LIN {X 0,Y 424.985,Z 1036.91,A -85,B 0,C 180,E1 -9892.159,E2 -9892.159} C_VEL
LIN {X 0,Y 424.826,Z 1042.69,A -85,B 0,C 180,E1 -9893.35,E2 -9893.35} C_VEL
LIN {X 0,Y 424.561,Z 1046.489,A -85,B 0,C 180,E1 -9894.3,E2 -9894.3} C_VEL
LIN {X 0,Y 424.338,Z 1049.56,A -85,B 0,C 180,E1 -9895.25,E2 -9895.25} C_VEL
LIN {X 0,Y 424.395,Z 1051.936,A -85,B 0,C 180,E1 -9896.202,E2 -9896.202} C_VEL
LIN {X 0,Y 424.27,Z 1053.752,A -85,B 0,C 180,E1 -9897.152,E2 -9897.152} C_VEL
LIN {X 0,Y 424.174,Z 1055.045,A -85,B 0,C 180,E1 -9898.101,E2 -9898.101} C_VEL
LIN {X 0,Y 424.113,Z 1055.839,A -85,B 0,C 180,E1 -9899.051,E2 -9899.051} C_VEL
LIN {X 0,Y 424.106,Z 1056.112,A -85,B 0,C 180,E1 -9900,E2 -9900} C_VEL
LIN {X 0,Y 424.112,Z 1055.78,A -85,B 0,C 180,E1 -9900.95,E2 -9900.95} C_VEL
LIN {X 0,Y 424.165,Z 1054.937,A -85,B 0,C 180,E1 -9901.899,E2 -9901.899} C_VEL
LIN {X 0,Y 424.262,Z 1053.59,A -85,B 0,C 180,E1 -9902.849,E2 -9902.849} C_VEL
LIN {X 0,Y 424.316,Z 1050.534,A -85,B 0,C 180,E1 -9904.275,E2 -9904.275} C_VEL
LIN {X 0,Y 424.525,Z 1046.159,A -85,B 0,C 180,E1 -9905.701,E2 -9905.701} C_VEL
LIN {X 0,Y 424.759,Z 1040.098,A -85,B 0,C 180,E1 -9907.128,E2 -9907.128} C_VEL
LIN {X 0,Y 424.953,Z 1035.048,A -85,B 0,C 180,E1 -9908.082,E2 -9908.082} C_VEL
LIN {X 0,Y 425.243,Z 1028.948,A -85,B 0,C 180,E1 -9909.034,E2 -9909.034} C_VEL
LIN {X 0,Y 425.687,Z 1020.492,A -85,B 0,C 180,E1 -9910.103,E2 -9910.103} C_VEL
LIN {X 0,Y 426.165,Z 1011.11,A -85,B 0,C 180,E1 -9911.053,E2 -9911.053} C_VEL
LIN {X 0,Y 426.592,Z 1000.255,A -85,B 0,C 180,E1 -9911.885,E2 -9911.885} C_VEL
LIN {X 0,Y 426.862,Z 991.105,A -85,B 0,C 180,E1 -9912.42,E2 -9912.42} C_VEL
LIN {X 0,Y 427.087,Z 981.57,A -85,B 0,C 180,E1 -9912.836,E2 -9912.836} C_VEL
LIN {X 0,Y 427.334,Z 971.535,A -85,B 0,C 180,E1 -9913.131,E2 -9913.131} C_VEL
LIN {X 0,Y 427.866,Z 911.953,A -85,B 0,C 180,E1 -9914.276,E2 -9914.276} C_VEL
LIN {X 0,Y 425.344,Z 897.558,A -85,B 0,C 180,E1 -9914.656,E2 -9914.656} C_VEL
LIN {X 0,Y 425.733,Z 888.265,A -85,B 0,C 180,E1 -9917.287,E2 -9917.287} C_VEL
LIN {X 0,Y 425.456,Z 882.672,A -85,B 0,C 180,E1 -9918.916,E2 -9918.916} C_VEL
LIN {X 0,Y 425.385,Z 882.313,A -85,B 0,C 180,E1 -9919.045,E2 -9919.045} C_VEL
LIN {X 0,Y 425.286,Z 882.318,A -85,B 0,C 180,E1 -9922.339,E2 -9922.339} C_VEL
LIN {X 0,Y 425.25,Z 882.327,A -85,B 0,C 180,E1 -9925.449,E2 -9925.449} C_VEL
LIN {X 0,Y 425.297,Z 882.318,A -85,B 0,C 180,E1 -9928.858,E2 -9928.858} C_VEL
LIN {X 0,Y 425.254,Z 882.324,A -85,B 0,C 180,E1 -9931.929,E2 -9931.929} C_VEL
LIN {X 0,Y 425.294,Z 882.32,A -85,B 0,C 180,E1 -9935.337,E2 -9935.337} C_VEL
LIN {X 0,Y 425.275,Z 882.319,A -85,B 0,C 180,E1 -9938.902,E2 -9938.902} C_VEL
LIN {X 0,Y 425.256,Z 882.322,A -85,B 0,C 180,E1 -9942.656,E2 -9942.656} C_VEL
LIN {X 0,Y 425.285,Z 882.318,A -85,B 0,C 180,E1 -9945.284,E2 -9945.284} C_VEL
LIN {X 0,Y 425.247,Z 882.326,A -85,B 0,C 180,E1 -9948.618,E2 -9948.618} C_VEL
LIN {X 0,Y 425.27,Z 882.326,A -85,B 0,C 180,E1 -9952.305,E2 -9952.305} C_VEL
LIN {X 0,Y 425.288,Z 882.318,A -85,B 0,C 180,E1 -9955.816,E2 -9955.816} C_VEL
LIN {X 0,Y 425.288,Z 882.319,A -85,B 0,C 180,E1 -9959.241,E2 -9959.241} C_VEL
LIN {X 0,Y 425.24,Z 882.326,A -85,B 0,C 180,E1 -9962.435,E2 -9962.435} C_VEL
LIN {X 0,Y 425.319,Z 882.315,A -85,B 0,C 180,E1 -9965.6,E2 -9965.6} C_VEL
LIN {X 0,Y 425.286,Z 882.32,A -85,B 0,C 180,E1 -9968.681,E2 -9968.681} C_VEL
LIN {X 0,Y 425.3,Z 882.318,A -85,B 0,C 180,E1 -9971.701,E2 -9971.701} C_VEL
LIN {X 0,Y 425.324,Z 882.314,A -85,B 0,C 180,E1 -9974.67,E2 -9974.67} C_VEL
LIN {X 0,Y 425.411,Z 882.309,A -85,B 0,C 180,E1 -9977.598,E2 -9977.598} C_VEL
LIN {X 0,Y 425.398,Z 882.308,A -85,B 0,C 180,E1 -9981.449,E2 -9981.449} C_VEL
LIN {X 0,Y 425.497,Z 882.293,A -85,B 0,C 180,E1 -9984.377,E2 -9984.377} C_VEL
LIN {X 0,Y 425.564,Z 882.289,A -85,B 0,C 180,E1 -9988.107,E2 -9988.107} C_VEL
LIN {X 0,Y 425.495,Z 882.293,A -85,B 0,C 180,E1 -9988.519,E2 -9988.519} C_VEL
LIN {X 0,Y 424.768,Z 882.383,A -85,B 0,C 180,E1 -9989.308,E2 -9989.308} C_VEL
LIN {X 0,Y 421.933,Z 882.737,A -85,B 0,C 180,E1 -9990.592,E2 -9990.592} C_VEL
LIN {X 0,Y 419.57,Z 883.031,A -85,B 0,C 180,E1 -9991.629,E2 -9991.629} C_VEL
LIN {X 0,Y 418.55,Z 883.161,A -85,B 0,C 180,E1 -9992.429,E2 -9992.429} C_VEL
LIN {X 0,Y 418.461,Z 883.168,A -85,B 0,C 180,E1 -9992.7,E2 -9992.7} C_VEL
LIN {X 0,Y 418.473,Z 883.168,A -85,B 0,C 180,E1 -9995.784,E2 -9995.784} C_VEL
LIN {X 0,Y 418.37,Z 883.184,A -85,B 0,C 180,E1 -9998.696,E2 -9998.696} C_VEL
LIN {X 0,Y 418.357,Z 883.188,A -85,B 0,C 180,E1 -10002.615,E2 -10002.615} C_VEL
LIN {X 0,Y 418.284,Z 883.195,A -85,B 0,C 180,E1 -10006.597,E2 -10006.597} C_VEL
LIN {X 0,Y 418.247,Z 883.195,A -85,B 0,C 180,E1 -10009.779,E2 -10009.779} C_VEL
LIN {X 0,Y 418.228,Z 883.2,A -85,B 0,C 180,E1 -10012.737,E2 -10012.737} C_VEL
LIN {X 0,Y 418.213,Z 883.199,A -85,B 0,C 180,E1 -10015.908,E2 -10015.908} C_VEL
LIN {X 0,Y 418.259,Z 883.198,A -85,B 0,C 180,E1 -10019.163,E2 -10019.163} C_VEL
LIN {X 0,Y 418.235,Z 883.196,A -85,B 0,C 180,E1 -10022.529,E2 -10022.529} C_VEL
LIN {X 0,Y 418.251,Z 883.195,A -85,B 0,C 180,E1 -10024.842,E2 -10024.842} C_VEL
LIN {X 0,Y 418.235,Z 883.197,A -85,B 0,C 180,E1 -10028.444,E2 -10028.444} C_VEL
LIN {X 0,Y 418.221,Z 883.202,A -85,B 0,C 180,E1 -10032.236,E2 -10032.236} C_VEL
LIN {X 0,Y 418.238,Z 883.196,A -85,B 0,C 180,E1 -10035.108,E2 -10035.108} C_VEL
LIN {X 0,Y 418.221,Z 883.2,A -85,B 0,C 180,E1 -10037.764,E2 -10037.764} C_VEL
LIN {X 0,Y 418.23,Z 883.197,A -85,B 0,C 180,E1 -10041.555,E2 -10041.555} C_VEL
LIN {X 0,Y 418.253,Z 883.195,A -85,B 0,C 180,E1 -10045.158,E2 -10045.158} C_VEL
LIN {X 0,Y 418.242,Z 883.195,A -85,B 0,C 180,E1 -10047.471,E2 -10047.471} C_VEL
LIN {X 0,Y 418.261,Z 883.199,A -85,B 0,C 180,E1 -10050.898,E2 -10050.898} C_VEL
LIN {X 0,Y 418.213,Z 883.199,A -85,B 0,C 180,E1 -10054.092,E2 -10054.092} C_VEL
LIN {X 0,Y 418.235,Z 883.198,A -85,B 0,C 180,E1 -10057.552,E2 -10057.552} C_VEL
LIN {X 0,Y 418.255,Z 883.194,A -85,B 0,C 180,E1 -10060.362,E2 -10060.362} C_VEL
LIN {X 0,Y 418.283,Z 883.197,A -85,B 0,C 180,E1 -10063.403,E2 -10063.403} C_VEL
LIN {X 0,Y 418.355,Z 883.187,A -85,B 0,C 180,E1 -10067.385,E2 -10067.385} C_VEL
LIN {X 0,Y 418.369,Z 883.182,A -85,B 0,C 180,E1 -10071.304,E2 -10071.304} C_VEL
LIN {X 0,Y 418.471,Z 883.169,A -85,B 0,C 180,E1 -10074.216,E2 -10074.216} C_VEL
LIN {X 0,Y 418.53,Z 883.165,A -85,B 0,C 180,E1 -10078.075,E2 -10078.075} C_VEL
LIN {X 0,Y 418.408,Z 883.175,A -85,B 0,C 180,E1 -10080.962,E2 -10080.962} C_VEL
LIN {X 0,Y 418.454,Z 883.169,A -85,B 0,C 180,E1 -10082.888,E2 -10082.888} C_VEL
LIN {X 0,Y 418.47,Z 883.168,A -85,B 0,C 180,E1 -10085.783,E2 -10085.783} C_VEL
LIN {X 0,Y 418.368,Z 883.184,A -85,B 0,C 180,E1 -10088.695,E2 -10088.695} C_VEL
LIN {X 0,Y 418.354,Z 883.189,A -85,B 0,C 180,E1 -10092.614,E2 -10092.614} C_VEL
LIN {X 0,Y 418.281,Z 883.195,A -85,B 0,C 180,E1 -10096.596,E2 -10096.596} C_VEL
LIN {X 0,Y 418.244,Z 883.195,A -85,B 0,C 180,E1 -10099.779,E2 -10099.779} C_VEL
LIN {X 0,Y 418.224,Z 883.201,A -85,B 0,C 180,E1 -10102.737,E2 -10102.737} C_VEL
LIN {X 0,Y 418.209,Z 883.2,A -85,B 0,C 180,E1 -10105.908,E2 -10105.908} C_VEL
LIN {X 0,Y 418.255,Z 883.199,A -85,B 0,C 180,E1 -10109.162,E2 -10109.162} C_VEL
LIN {X 0,Y 418.23,Z 883.197,A -85,B 0,C 180,E1 -10112.529,E2 -10112.529} C_VEL
LIN {X 0,Y 418.247,Z 883.195,A -85,B 0,C 180,E1 -10114.842,E2 -10114.842} C_VEL
LIN {X 0,Y 418.23,Z 883.197,A -85,B 0,C 180,E1 -10118.444,E2 -10118.444} C_VEL
LIN {X 0,Y 418.216,Z 883.202,A -85,B 0,C 180,E1 -10122.236,E2 -10122.236} C_VEL
LIN {X 0,Y 418.233,Z 883.196,A -85,B 0,C 180,E1 -10125.108,E2 -10125.108} C_VEL
LIN {X 0,Y 418.216,Z 883.201,A -85,B 0,C 180,E1 -10127.763,E2 -10127.763} C_VEL
LIN {X 0,Y 418.225,Z 883.198,A -85,B 0,C 180,E1 -10131.555,E2 -10131.555} C_VEL
LIN {X 0,Y 418.248,Z 883.195,A -85,B 0,C 180,E1 -10135.158,E2 -10135.158} C_VEL
LIN {X 0,Y 418.238,Z 883.196,A -85,B 0,C 180,E1 -10137.471,E2 -10137.471} C_VEL
LIN {X 0,Y 418.256,Z 883.199,A -85,B 0,C 180,E1 -10140.898,E2 -10140.898} C_VEL
LIN {X 0,Y 418.258,Z 883.255,A -85,B 0,C 180,E1 -10144.411,E2 -10144.411} C_VEL
LIN {X 0,Y 420.166,Z 893.538,A -85,B 0,C 180,E1 -10146.921,E2 -10146.921} C_VEL
LIN {X 0,Y 419.942,Z 901.074,A -85,B 0,C 180,E1 -10148.654,E2 -10148.654} C_VEL
LIN {X 0,Y 419.121,Z 915.553,A -85,B 0,C 180,E1 -10151.928,E2 -10151.928} C_VEL
LIN {X 0,Y 418.376,Z 930.113,A -85,B 0,C 180,E1 -10155.141,E2 -10155.141} C_VEL
LIN {X 0,Y 420.95,Z 951.978,A -85,B 0,C 180,E1 -10155.663,E2 -10155.663} C_VEL
LIN {X 0,Y 420.299,Z 1007.525,A -85,B 0,C 180,E1 -10156.769,E2 -10156.769} C_VEL
LIN {X 0,Y 419.904,Z 1018.346,A -85,B 0,C 180,E1 -10157.125,E2 -10157.125} C_VEL
LIN {X 0,Y 419.54,Z 1029.214,A -85,B 0,C 180,E1 -10157.667,E2 -10157.667} C_VEL
LIN {X 0,Y 419.115,Z 1039.643,A -85,B 0,C 180,E1 -10158.391,E2 -10158.391} C_VEL
LIN {X 0,Y 418.722,Z 1047.891,A -85,B 0,C 180,E1 -10159.116,E2 -10159.116} C_VEL
LIN {X 0,Y 418.32,Z 1055.741,A -85,B 0,C 180,E1 -10159.962,E2 -10159.962} C_VEL
LIN {X 0,Y 417.897,Z 1063.972,A -85,B 0,C 180,E1 -10161.05,E2 -10161.05} C_VEL
LIN {X 0,Y 417.593,Z 1071.163,A -85,B 0,C 180,E1 -10162.262,E2 -10162.262} C_VEL
LIN {X 0,Y 417.341,Z 1076.904,A -85,B 0,C 180,E1 -10163.49,E2 -10163.49} C_VEL
LIN {X 0,Y 417.213,Z 1081.322,A -85,B 0,C 180,E1 -10164.684,E2 -10164.684} C_VEL
LIN {X 0,Y 417.114,Z 1084.17,A -85,B 0,C 180,E1 -10165.651,E2 -10165.651} C_VEL
LIN {X 0,Y 417.086,Z 1087.252,A -85,B 0,C 180,E1 -10167.102,E2 -10167.102} C_VEL
LIN {X 0,Y 417.073,Z 1088.619,A -85,B 0,C 180,E1 -10168.068,E2 -10168.068} C_VEL
LIN {X 0,Y 417.029,Z 1089.473,A -85,B 0,C 180,E1 -10169.034,E2 -10169.034} C_VEL
LIN {X 0,Y 417.023,Z 1089.769,A -85,B 0,C 180,E1 -10170,E2 -10170} C_VEL
LIN {X 0,Y 417.029,Z 1089.463,A -85,B 0,C 180,E1 -10170.965,E2 -10170.965} C_VEL
LIN {X 0,Y 417.073,Z 1088.655,A -85,B 0,C 180,E1 -10171.931,E2 -10171.931} C_VEL
LIN {X 0,Y 417.082,Z 1087.336,A -85,B 0,C 180,E1 -10172.897,E2 -10172.897} C_VEL
LIN {X 0,Y 417.114,Z 1084.266,A -85,B 0,C 180,E1 -10174.348,E2 -10174.348} C_VEL
LIN {X 0,Y 417.214,Z 1081.472,A -85,B 0,C 180,E1 -10175.316,E2 -10175.316} C_VEL
LIN {X 0,Y 417.342,Z 1077.084,A -85,B 0,C 180,E1 -10176.511,E2 -10176.511} C_VEL
LIN {X 0,Y 417.524,Z 1072.603,A -85,B 0,C 180,E1 -10177.496,E2 -10177.496} C_VEL
LIN {X 0,Y 417.725,Z 1067.312,A -85,B 0,C 180,E1 -10178.465,E2 -10178.465} C_VEL
LIN {X 0,Y 418.117,Z 1060.957,A -85,B 0,C 180,E1 -10179.432,E2 -10179.432} C_VEL
LIN {X 0,Y 418.516,Z 1053.237,A -85,B 0,C 180,E1 -10180.4,E2 -10180.4} C_VEL
LIN {X 0,Y 419.023,Z 1043.686,A -85,B 0,C 180,E1 -10181.366,E2 -10181.366} C_VEL
LIN {X 0,Y 419.428,Z 1034.458,A -85,B 0,C 180,E1 -10182.09,E2 -10182.09} C_VEL
LIN {X 0,Y 419.811,Z 1024.464,A -85,B 0,C 180,E1 -10182.693,E2 -10182.693} C_VEL
LIN {X 0,Y 420.227,Z 1015.136,A -85,B 0,C 180,E1 -10183.11,E2 -10183.11} C_VEL
LIN {X 0,Y 420.542,Z 1005.59,A -85,B 0,C 180,E1 -10183.407,E2 -10183.407} C_VEL
LIN {X 0,Y 421.166,Z 949.616,A -85,B 0,C 180,E1 -10184.57,E2 -10184.57} C_VEL
LIN {X 0,Y 418.931,Z 931.747,A -85,B 0,C 180,E1 -10185.066,E2 -10185.066} C_VEL
LIN {X 0,Y 418.429,Z 928.431,A -85,B 0,C 180,E1 -10185.177,E2 -10185.177} C_VEL
LIN {X 0,Y 419.239,Z 913.478,A -85,B 0,C 180,E1 -10188.573,E2 -10188.573} C_VEL
LIN {X 0,Y 420.175,Z 899.489,A -85,B 0,C 180,E1 -10191.849,E2 -10191.849} C_VEL
LIN {X 0,Y 420.291,Z 894.287,A -85,B 0,C 180,E1 -10193.119,E2 -10193.119} C_VEL
LIN {X 0,Y 418.805,Z 885.701,A -85,B 0,C 180,E1 -10195.403,E2 -10195.403} C_VEL
LIN {X 0,Y 418.244,Z 883.203,A -85,B 0,C 180,E1 -10196.174,E2 -10196.174} C_VEL
LIN {X 0,Y 418.252,Z 883.202,A -85,B 0,C 180,E1 -10199.163,E2 -10199.163} C_VEL
LIN {X 0,Y 418.246,Z 883.202,A -85,B 0,C 180,E1 -10202.842,E2 -10202.842} C_VEL
LIN {X 0,Y 418.235,Z 883.199,A -85,B 0,C 180,E1 -10206.236,E2 -10206.236} C_VEL
LIN {X 0,Y 418.19,Z 883.208,A -85,B 0,C 180,E1 -10209.689,E2 -10209.689} C_VEL
LIN {X 0,Y 418.203,Z 883.204,A -85,B 0,C 180,E1 -10212.318,E2 -10212.318} C_VEL
LIN {X 0,Y 418.232,Z 883.199,A -85,B 0,C 180,E1 -10215.108,E2 -10215.108} C_VEL
LIN {X 0,Y 418.214,Z 883.203,A -85,B 0,C 180,E1 -10217.764,E2 -10217.764} C_VEL
LIN {X 0,Y 418.224,Z 883.201,A -85,B 0,C 180,E1 -10221.555,E2 -10221.555} C_VEL
LIN {X 0,Y 418.247,Z 883.197,A -85,B 0,C 180,E1 -10225.158,E2 -10225.158} C_VEL
LIN {X 0,Y 418.237,Z 883.199,A -85,B 0,C 180,E1 -10227.472,E2 -10227.472} C_VEL
LIN {X 0,Y 418.255,Z 883.2,A -85,B 0,C 180,E1 -10230.899,E2 -10230.899} C_VEL
LIN {X 0,Y 418.207,Z 883.204,A -85,B 0,C 180,E1 -10234.092,E2 -10234.092} C_VEL
LIN {X 0,Y 418.229,Z 883.206,A -85,B 0,C 180,E1 -10237.553,E2 -10237.553} C_VEL
LIN {X 0,Y 418.265,Z 883.342,A -85,B 0,C 180,E1 -10239.689,E2 -10239.689} C_VEL
LIN {X 0,Y 419.149,Z 888.393,A -85,B 0,C 180,E1 -10241.423,E2 -10241.423} C_VEL
LIN {X 0,Y 419.053,Z 894.734,A -85,B 0,C 180,E1 -10243.435,E2 -10243.435} C_VEL
LIN {X 0,Y 418.734,Z 899.597,A -85,B 0,C 180,E1 -10244.928,E2 -10244.928} C_VEL
LIN {X 0,Y 421.443,Z 912.992,A -85,B 0,C 180,E1 -10245.358,E2 -10245.358} C_VEL
LIN {X 0,Y 420.863,Z 963.311,A -85,B 0,C 180,E1 -10246.415,E2 -10246.415} C_VEL
LIN {X 0,Y 420.498,Z 978.918,A -85,B 0,C 180,E1 -10246.776,E2 -10246.776} C_VEL
LIN {X 0,Y 420.228,Z 990.494,A -85,B 0,C 180,E1 -10247.259,E2 -10247.259} C_VEL
LIN {X 0,Y 419.889,Z 998.061,A -85,B 0,C 180,E1 -10247.678,E2 -10247.678} C_VEL
LIN {X 0,Y 419.592,Z 1006.59,A -85,B 0,C 180,E1 -10248.283,E2 -10248.283} C_VEL
LIN {X 0,Y 419.251,Z 1014.804,A -85,B 0,C 180,E1 -10249.008,E2 -10249.008} C_VEL
LIN {X 0,Y 418.832,Z 1022.619,A -85,B 0,C 180,E1 -10249.852,E2 -10249.852} C_VEL
LIN {X 0,Y 418.373,Z 1029.936,A -85,B 0,C 180,E1 -10250.818,E2 -10250.818} C_VEL
LIN {X 0,Y 417.969,Z 1037.324,A -85,B 0,C 180,E1 -10252.027,E2 -10252.027} C_VEL
LIN {X 0,Y 417.763,Z 1043.07,A -85,B 0,C 180,E1 -10253.238,E2 -10253.238} C_VEL
LIN {X 0,Y 417.527,Z 1046.849,A -85,B 0,C 180,E1 -10254.204,E2 -10254.204} C_VEL
LIN {X 0,Y 417.272,Z 1049.911,A -85,B 0,C 180,E1 -10255.17,E2 -10255.17} C_VEL
LIN {X 0,Y 417.314,Z 1052.278,A -85,B 0,C 180,E1 -10256.138,E2 -10256.138} C_VEL
LIN {X 0,Y 417.21,Z 1054.083,A -85,B 0,C 180,E1 -10257.104,E2 -10257.104} C_VEL
LIN {X 0,Y 417.102,Z 1055.363,A -85,B 0,C 180,E1 -10258.069,E2 -10258.069} C_VEL
LIN {X 0,Y 417.034,Z 1056.141,A -85,B 0,C 180,E1 -10259.035,E2 -10259.035} C_VEL
LIN {X 0,Y 417.025,Z 1056.403,A -85,B 0,C 180,E1 -10260,E2 -10260} C_VEL
LIN {X 0,Y 417.033,Z 1056.058,A -85,B 0,C 180,E1 -10260.966,E2 -10260.966} C_VEL
LIN {X 0,Y 417.093,Z 1055.187,A -85,B 0,C 180,E1 -10261.932,E2 -10261.932} C_VEL
LIN {X 0,Y 417.181,Z 1053.815,A -85,B 0,C 180,E1 -10262.897,E2 -10262.897} C_VEL
LIN {X 0,Y 417.226,Z 1050.717,A -85,B 0,C 180,E1 -10264.348,E2 -10264.348} C_VEL
LIN {X 0,Y 417.464,Z 1046.294,A -85,B 0,C 180,E1 -10265.798,E2 -10265.798} C_VEL
LIN {X 0,Y 417.697,Z 1040.156,A -85,B 0,C 180,E1 -10267.25,E2 -10267.25} C_VEL
LIN {X 0,Y 417.906,Z 1035.047,A -85,B 0,C 180,E1 -10268.219,E2 -10268.219} C_VEL
LIN {X 0,Y 418.233,Z 1028.882,A -85,B 0,C 180,E1 -10269.186,E2 -10269.186} C_VEL
LIN {X 0,Y 418.626,Z 1021.379,A -85,B 0,C 180,E1 -10270.153,E2 -10270.153} C_VEL
LIN {X 0,Y 419.071,Z 1013.359,A -85,B 0,C 180,E1 -10270.998,E2 -10270.998} C_VEL
LIN {X 0,Y 419.502,Z 1003.366,A -85,B 0,C 180,E1 -10271.843,E2 -10271.843} C_VEL
LIN {X 0,Y 419.796,Z 992.781,A -85,B 0,C 180,E1 -10272.509,E2 -10272.509} C_VEL
LIN {X 0,Y 420.046,Z 982.95,A -85,B 0,C 180,E1 -10272.963,E2 -10272.963} C_VEL
LIN {X 0,Y 420.314,Z 973.531,A -85,B 0,C 180,E1 -10273.262,E2 -10273.262} C_VEL
LIN {X 0,Y 420.965,Z 912.92,A -85,B 0,C 180,E1 -10274.463,E2 -10274.463} C_VEL
LIN {X 0,Y 418.335,Z 897.792,A -85,B 0,C 180,E1 -10274.876,E2 -10274.876} C_VEL
LIN {X 0,Y 418.721,Z 888.371,A -85,B 0,C 180,E1 -10277.586,E2 -10277.586} C_VEL
LIN {X 0,Y 418.349,Z 883.188,A -85,B 0,C 180,E1 -10279.187,E2 -10279.187} C_VEL
LIN {X 0,Y 418.225,Z 883.201,A -85,B 0,C 180,E1 -10282.738,E2 -10282.738} C_VEL
LIN {X 0,Y 418.21,Z 883.2,A -85,B 0,C 180,E1 -10285.909,E2 -10285.909} C_VEL
LIN {X 0,Y 418.256,Z 883.198,A -85,B 0,C 180,E1 -10289.163,E2 -10289.163} C_VEL
LIN {X 0,Y 418.25,Z 883.195,A -85,B 0,C 180,E1 -10292.842,E2 -10292.842} C_VEL
LIN {X 0,Y 418.24,Z 883.197,A -85,B 0,C 180,E1 -10296.237,E2 -10296.237} C_VEL
LIN {X 0,Y 418.199,Z 883.206,A -85,B 0,C 180,E1 -10299.689,E2 -10299.689} C_VEL
LIN {X 0,Y 418.207,Z 883.203,A -85,B 0,C 180,E1 -10302.318,E2 -10302.318} C_VEL
LIN {X 0,Y 418.236,Z 883.196,A -85,B 0,C 180,E1 -10305.109,E2 -10305.109} C_VEL
LIN {X 0,Y 418.219,Z 883.2,A -85,B 0,C 180,E1 -10307.764,E2 -10307.764} C_VEL
LIN {X 0,Y 418.229,Z 883.197,A -85,B 0,C 180,E1 -10311.556,E2 -10311.556} C_VEL
LIN {X 0,Y 418.252,Z 883.195,A -85,B 0,C 180,E1 -10315.158,E2 -10315.158} C_VEL
LIN {X 0,Y 418.242,Z 883.196,A -85,B 0,C 180,E1 -10317.472,E2 -10317.472} C_VEL
LIN {X 0,Y 418.26,Z 883.199,A -85,B 0,C 180,E1 -10320.899,E2 -10320.899} C_VEL
LIN {X 0,Y 418.213,Z 883.199,A -85,B 0,C 180,E1 -10324.092,E2 -10324.092} C_VEL
LIN {X 0,Y 418.228,Z 883.202,A -85,B 0,C 180,E1 -10327.263,E2 -10327.263} C_VEL
LIN {X 0,Y 418.255,Z 883.194,A -85,B 0,C 180,E1 -10330.363,E2 -10330.363} C_VEL
LIN {X 0,Y 418.33,Z 883.191,A -85,B 0,C 180,E1 -10333.405,E2 -10333.405} C_VEL
LIN {X 0,Y 418.357,Z 883.187,A -85,B 0,C 180,E1 -10337.386,E2 -10337.386} C_VEL
LIN {X 0,Y 418.37,Z 883.182,A -85,B 0,C 180,E1 -10341.304,E2 -10341.304} C_VEL
LIN {X 0,Y 418.473,Z 883.169,A -85,B 0,C 180,E1 -10344.217,E2 -10344.217} C_VEL
LIN {X 0,Y 418.532,Z 883.165,A -85,B 0,C 180,E1 -10348.076,E2 -10348.076} C_VEL
LIN {X 0,Y 418.41,Z 883.174,A -85,B 0,C 180,E1 -10350.963,E2 -10350.963} C_VEL
LIN {X 0,Y 418.461,Z 883.168,A -85,B 0,C 180,E1 -10352.7,E2 -10352.7} C_VEL
LIN {X 0,Y 417.781,Z 883.254,A -85,B 0,C 180,E1 -10353.502,E2 -10353.502} C_VEL
LIN {X 0,Y 414.933,Z 883.613,A -85,B 0,C 180,E1 -10354.806,E2 -10354.806} C_VEL
LIN {X 0,Y 412.524,Z 883.913,A -85,B 0,C 180,E1 -10355.859,E2 -10355.859} C_VEL
LIN {X 0,Y 411.482,Z 884.042,A -85,B 0,C 180,E1 -10356.672,E2 -10356.672} C_VEL
LIN {X 0,Y 411.391,Z 884.05,A -85,B 0,C 180,E1 -10356.948,E2 -10356.948} C_VEL
LIN {X 0,Y 411.276,Z 884.064,A -85,B 0,C 180,E1 -10359.839,E2 -10359.839} C_VEL
LIN {X 0,Y 411.31,Z 884.061,A -85,B 0,C 180,E1 -10363.103,E2 -10363.103} C_VEL
LIN {X 0,Y 411.214,Z 884.077,A -85,B 0,C 180,E1 -10366.891,E2 -10366.891} C_VEL
LIN {X 0,Y 411.209,Z 884.072,A -85,B 0,C 180,E1 -10369.988,E2 -10369.988} C_VEL
LIN {X 0,Y 411.179,Z 884.082,A -85,B 0,C 180,E1 -10373.149,E2 -10373.149} C_VEL
LIN {X 0,Y 411.167,Z 884.077,A -85,B 0,C 180,E1 -10376.386,E2 -10376.386} C_VEL
LIN {X 0,Y 411.196,Z 884.076,A -85,B 0,C 180,E1 -10379.713,E2 -10379.713} C_VEL
LIN {X 0,Y 411.207,Z 884.074,A -85,B 0,C 180,E1 -10383.156,E2 -10383.156} C_VEL
LIN {X 0,Y 411.191,Z 884.074,A -85,B 0,C 180,E1 -10386.551,E2 -10386.551} C_VEL
LIN {X 0,Y 411.17,Z 884.082,A -85,B 0,C 180,E1 -10389.72,E2 -10389.72} C_VEL
LIN {X 0,Y 411.164,Z 884.077,A -85,B 0,C 180,E1 -10393.135,E2 -10393.135} C_VEL
LIN {X 0,Y 411.167,Z 884.081,A -85,B 0,C 180,E1 -10395.882,E2 -10395.882} C_VEL
LIN {X 0,Y 411.159,Z 884.078,A -85,B 0,C 180,E1 -10399.492,E2 -10399.492} C_VEL
LIN {X 0,Y 411.18,Z 884.078,A -85,B 0,C 180,E1 -10402.024,E2 -10402.024} C_VEL
LIN {X 0,Y 411.205,Z 884.073,A -85,B 0,C 180,E1 -10405.123,E2 -10405.123} C_VEL
LIN {X 0,Y 411.163,Z 884.078,A -85,B 0,C 180,E1 -10408.002,E2 -10408.002} C_VEL
LIN {X 0,Y 411.171,Z 884.077,A -85,B 0,C 180,E1 -10411.406,E2 -10411.406} C_VEL
LIN {X 0,Y 411.191,Z 884.081,A -85,B 0,C 180,E1 -10414.941,E2 -10414.941} C_VEL
LIN {X 0,Y 411.203,Z 884.072,A -85,B 0,C 180,E1 -10417.913,E2 -10417.913} C_VEL
LIN {X 0,Y 411.193,Z 884.079,A -85,B 0,C 180,E1 -10421.049,E2 -10421.049} C_VEL
LIN {X 0,Y 411.202,Z 884.072,A -85,B 0,C 180,E1 -10424.129,E2 -10424.129} C_VEL
LIN {X 0,Y 411.305,Z 884.063,A -85,B 0,C 180,E1 -10427.165,E2 -10427.165} C_VEL
LIN {X 0,Y 411.274,Z 884.065,A -85,B 0,C 180,E1 -10430.16,E2 -10430.16} C_VEL
LIN {X 0,Y 411.393,Z 884.049,A -85,B 0,C 180,E1 -10433.131,E2 -10433.131} C_VEL
LIN {X 0,Y 411.283,Z 884.063,A -85,B 0,C 180,E1 -10435.098,E2 -10435.098} C_VEL
LIN {X 0,Y 411.499,Z 884.042,A -85,B 0,C 180,E1 -10438.042,E2 -10438.042} C_VEL
LIN {X 0,Y 411.378,Z 884.05,A -85,B 0,C 180,E1 -10440.978,E2 -10440.978} C_VEL
LIN {X 0,Y 411.413,Z 884.046,A -85,B 0,C 180,E1 -10442.937,E2 -10442.937} C_VEL
LIN {X 0,Y 411.418,Z 884.048,A -85,B 0,C 180,E1 -10445.882,E2 -10445.882} C_VEL
LIN {X 0,Y 411.307,Z 884.062,A -85,B 0,C 180,E1 -10448.846,E2 -10448.846} C_VEL
LIN {X 0,Y 411.271,Z 884.064,A -85,B 0,C 180,E1 -10451.833,E2 -10451.833} C_VEL
LIN {X 0,Y 411.212,Z 884.076,A -85,B 0,C 180,E1 -10454.854,E2 -10454.854} C_VEL
LIN {X 0,Y 411.204,Z 884.072,A -85,B 0,C 180,E1 -10457.917,E2 -10457.917} C_VEL
LIN {X 0,Y 411.188,Z 884.081,A -85,B 0,C 180,E1 -10461.034,E2 -10461.034} C_VEL
LIN {X 0,Y 411.172,Z 884.076,A -85,B 0,C 180,E1 -10464.218,E2 -10464.218} C_VEL
LIN {X 0,Y 411.141,Z 884.084,A -85,B 0,C 180,E1 -10467.486,E2 -10467.486} C_VEL
LIN {X 0,Y 411.192,Z 884.076,A -85,B 0,C 180,E1 -10469.713,E2 -10469.713} C_VEL
LIN {X 0,Y 411.203,Z 884.075,A -85,B 0,C 180,E1 -10473.156,E2 -10473.156} C_VEL
LIN {X 0,Y 411.187,Z 884.074,A -85,B 0,C 180,E1 -10476.551,E2 -10476.551} C_VEL
LIN {X 0,Y 411.166,Z 884.083,A -85,B 0,C 180,E1 -10479.719,E2 -10479.719} C_VEL
LIN {X 0,Y 411.16,Z 884.078,A -85,B 0,C 180,E1 -10483.135,E2 -10483.135} C_VEL
LIN {X 0,Y 411.163,Z 884.082,A -85,B 0,C 180,E1 -10485.881,E2 -10485.881} C_VEL
LIN {X 0,Y 411.155,Z 884.078,A -85,B 0,C 180,E1 -10489.492,E2 -10489.492} C_VEL
LIN {X 0,Y 411.176,Z 884.079,A -85,B 0,C 180,E1 -10492.024,E2 -10492.024} C_VEL
LIN {X 0,Y 411.2,Z 884.073,A -85,B 0,C 180,E1 -10495.123,E2 -10495.123} C_VEL
LIN {X 0,Y 411.158,Z 884.079,A -85,B 0,C 180,E1 -10498.002,E2 -10498.002} C_VEL
LIN {X 0,Y 411.166,Z 884.078,A -85,B 0,C 180,E1 -10501.406,E2 -10501.406} C_VEL
LIN {X 0,Y 411.25,Z 884.212,A -85,B 0,C 180,E1 -10504.267,E2 -10504.267} C_VEL
LIN {X 0,Y 413.189,Z 895.116,A -85,B 0,C 180,E1 -10506.97,E2 -10506.97} C_VEL
LIN {X 0,Y 412.837,Z 904.062,A -85,B 0,C 180,E1 -10509.053,E2 -10509.053} C_VEL
LIN {X 0,Y 411.911,Z 919.423,A -85,B 0,C 180,E1 -10512.576,E2 -10512.576} C_VEL
LIN {X 0,Y 411.371,Z 929.893,A -85,B 0,C 180,E1 -10514.914,E2 -10514.914} C_VEL
LIN {X 0,Y 414.008,Z 951.851,A -85,B 0,C 180,E1 -10515.459,E2 -10515.459} C_VEL
LIN {X 0,Y 413.32,Z 1007.783,A -85,B 0,C 180,E1 -10516.604,E2 -10516.604} C_VEL
LIN {X 0,Y 412.901,Z 1018.405,A -85,B 0,C 180,E1 -10516.966,E2 -10516.966} C_VEL
LIN {X 0,Y 412.486,Z 1030.062,A -85,B 0,C 180,E1 -10517.578,E2 -10517.578} C_VEL
LIN {X 0,Y 412.104,Z 1038.763,A -85,B 0,C 180,E1 -10518.191,E2 -10518.191} C_VEL
LIN {X 0,Y 411.72,Z 1047.122,A -85,B 0,C 180,E1 -10518.928,E2 -10518.928} C_VEL
LIN {X 0,Y 411.264,Z 1055.055,A -85,B 0,C 180,E1 -10519.787,E2 -10519.787} C_VEL
LIN {X 0,Y 410.962,Z 1061.627,A -85,B 0,C 180,E1 -10520.65,E2 -10520.65} C_VEL
LIN {X 0,Y 410.617,Z 1067.88,A -85,B 0,C 180,E1 -10521.635,E2 -10521.635} C_VEL
LIN {X 0,Y 410.383,Z 1074.269,A -85,B 0,C 180,E1 -10522.868,E2 -10522.868} C_VEL
LIN {X 0,Y 410.14,Z 1079.307,A -85,B 0,C 180,E1 -10524.099,E2 -10524.099} C_VEL
LIN {X 0,Y 410.043,Z 1083.793,A -85,B 0,C 180,E1 -10525.576,E2 -10525.576} C_VEL
LIN {X 0,Y 409.987,Z 1086.908,A -85,B 0,C 180,E1 -10527.052,E2 -10527.052} C_VEL
LIN {X 0,Y 410.003,Z 1088.3,A -85,B 0,C 180,E1 -10528.035,E2 -10528.035} C_VEL
LIN {X 0,Y 409.953,Z 1089.175,A -85,B 0,C 180,E1 -10529.018,E2 -10529.018} C_VEL
LIN {X 0,Y 409.945,Z 1089.474,A -85,B 0,C 180,E1 -10530,E2 -10530} C_VEL
LIN {X 0,Y 409.953,Z 1089.178,A -85,B 0,C 180,E1 -10530.982,E2 -10530.982} C_VEL
LIN {X 0,Y 410.002,Z 1088.381,A -85,B 0,C 180,E1 -10531.964,E2 -10531.964} C_VEL
LIN {X 0,Y 409.981,Z 1087.071,A -85,B 0,C 180,E1 -10532.948,E2 -10532.948} C_VEL
LIN {X 0,Y 410.043,Z 1084.017,A -85,B 0,C 180,E1 -10534.423,E2 -10534.423} C_VEL
LIN {X 0,Y 410.134,Z 1081.238,A -85,B 0,C 180,E1 -10535.408,E2 -10535.408} C_VEL
LIN {X 0,Y 410.237,Z 1077.488,A -85,B 0,C 180,E1 -10536.472,E2 -10536.472} C_VEL
LIN {X 0,Y 410.485,Z 1072.419,A -85,B 0,C 180,E1 -10537.625,E2 -10537.625} C_VEL
LIN {X 0,Y 410.784,Z 1065.676,A -85,B 0,C 180,E1 -10538.857,E2 -10538.857} C_VEL
LIN {X 0,Y 411.308,Z 1057.243,A -85,B 0,C 180,E1 -10540.087,E2 -10540.087} C_VEL
LIN {X 0,Y 411.768,Z 1048.595,A -85,B 0,C 180,E1 -10541.07,E2 -10541.07} C_VEL
LIN {X 0,Y 412.168,Z 1040.653,A -85,B 0,C 180,E1 -10541.807,E2 -10541.807} C_VEL
LIN {X 0,Y 412.536,Z 1032.553,A -85,B 0,C 180,E1 -10542.42,E2 -10542.42} C_VEL
LIN {X 0,Y 412.935,Z 1023.323,A -85,B 0,C 180,E1 -10542.97,E2 -10542.97} C_VEL
LIN {X 0,Y 413.393,Z 1013.797,A -85,B 0,C 180,E1 -10543.393,E2 -10543.393} C_VEL
LIN {X 0,Y 413.748,Z 1002.761,A -85,B 0,C 180,E1 -10543.726,E2 -10543.726} C_VEL
LIN {X 0,Y 414.416,Z 950.605,A -85,B 0,C 180,E1 -10544.839,E2 -10544.839} C_VEL
LIN {X 0,Y 412.121,Z 932.153,A -85,B 0,C 180,E1 -10545.369,E2 -10545.369} C_VEL
LIN {X 0,Y 411.484,Z 928.083,A -85,B 0,C 180,E1 -10545.51,E2 -10545.51} C_VEL
LIN {X 0,Y 412.407,Z 912.443,A -85,B 0,C 180,E1 -10549.15,E2 -10549.15} C_VEL
LIN {X 0,Y 413.26,Z 900.714,A -85,B 0,C 180,E1 -10551.971,E2 -10551.971} C_VEL
LIN {X 0,Y 413.472,Z 896.512,A -85,B 0,C 180,E1 -10553.013,E2 -10553.013} C_VEL
LIN {X 0,Y 412.061,Z 888.059,A -85,B 0,C 180,E1 -10555.318,E2 -10555.318} C_VEL
LIN {X 0,Y 411.198,Z 884.082,A -85,B 0,C 180,E1 -10556.515,E2 -10556.515} C_VEL
LIN {X 0,Y 411.19,Z 884.08,A -85,B 0,C 180,E1 -10559.713,E2 -10559.713} C_VEL
LIN {X 0,Y 411.202,Z 884.08,A -85,B 0,C 180,E1 -10563.156,E2 -10563.156} C_VEL
LIN {X 0,Y 411.185,Z 884.076,A -85,B 0,C 180,E1 -10566.551,E2 -10566.551} C_VEL
LIN {X 0,Y 411.16,Z 884.084,A -85,B 0,C 180,E1 -10569.719,E2 -10569.719} C_VEL
LIN {X 0,Y 411.159,Z 884.081,A -85,B 0,C 180,E1 -10573.135,E2 -10573.135} C_VEL
LIN {X 0,Y 411.16,Z 884.083,A -85,B 0,C 180,E1 -10575.882,E2 -10575.882} C_VEL
LIN {X 0,Y 411.153,Z 884.081,A -85,B 0,C 180,E1 -10579.493,E2 -10579.493} C_VEL
LIN {X 0,Y 411.174,Z 884.08,A -85,B 0,C 180,E1 -10582.024,E2 -10582.024} C_VEL
LIN {X 0,Y 411.199,Z 884.075,A -85,B 0,C 180,E1 -10585.124,E2 -10585.124} C_VEL
LIN {X 0,Y 411.157,Z 884.083,A -85,B 0,C 180,E1 -10588.002,E2 -10588.002} C_VEL
LIN {X 0,Y 411.165,Z 884.08,A -85,B 0,C 180,E1 -10591.406,E2 -10591.406} C_VEL
LIN {X 0,Y 411.186,Z 884.084,A -85,B 0,C 180,E1 -10594.942,E2 -10594.942} C_VEL
LIN {X 0,Y 411.197,Z 884.081,A -85,B 0,C 180,E1 -10597.913,E2 -10597.913} C_VEL
LIN {X 0,Y 411.21,Z 884.21,A -85,B 0,C 180,E1 -10599.36,E2 -10599.36} C_VEL
LIN {X 0,Y 412.267,Z 890.66,A -85,B 0,C 180,E1 -10601.617,E2 -10601.617} C_VEL
LIN {X 0,Y 412.043,Z 896.997,A -85,B 0,C 180,E1 -10603.655,E2 -10603.655} C_VEL
LIN {X 0,Y 411.84,Z 900.167,A -85,B 0,C 180,E1 -10604.607,E2 -10604.607} C_VEL
LIN {X 0,Y 414.63,Z 913.279,A -85,B 0,C 180,E1 -10605.051,E2 -10605.051} C_VEL
LIN {X 0,Y 414.769,Z 918.838,A -85,B 0,C 180,E1 -10605.183,E2 -10605.183} C_VEL
LIN {X 0,Y 413.751,Z 977.161,A -85,B 0,C 180,E1 -10606.462,E2 -10606.462} C_VEL
LIN {X 0,Y 413.413,Z 989.021,A -85,B 0,C 180,E1 -10606.92,E2 -10606.92} C_VEL
LIN {X 0,Y 412.995,Z 998.765,A -85,B 0,C 180,E1 -10607.469,E2 -10607.469} C_VEL
LIN {X 0,Y 412.669,Z 1007.182,A -85,B 0,C 180,E1 -10608.083,E2 -10608.083} C_VEL
LIN {X 0,Y 412.314,Z 1015.328,A -85,B 0,C 180,E1 -10608.821,E2 -10608.821} C_VEL
LIN {X 0,Y 411.876,Z 1023.118,A -85,B 0,C 180,E1 -10609.679,E2 -10609.679} C_VEL
LIN {X 0,Y 411.294,Z 1032.08,A -85,B 0,C 180,E1 -10610.906,E2 -10610.906} C_VEL
LIN {X 0,Y 410.889,Z 1038.968,A -85,B 0,C 180,E1 -10612.136,E2 -10612.136} C_VEL
LIN {X 0,Y 410.711,Z 1043.494,A -85,B 0,C 180,E1 -10613.121,E2 -10613.121} C_VEL
LIN {X 0,Y 410.494,Z 1047.255,A -85,B 0,C 180,E1 -10614.104,E2 -10614.104} C_VEL
LIN {X 0,Y 410.211,Z 1050.313,A -85,B 0,C 180,E1 -10615.086,E2 -10615.086} C_VEL
LIN {X 0,Y 410.235,Z 1052.667,A -85,B 0,C 180,E1 -10616.071,E2 -10616.071} C_VEL
LIN {X 0,Y 410.151,Z 1054.442,A -85,B 0,C 180,E1 -10617.054,E2 -10617.054} C_VEL
LIN {X 0,Y 410.033,Z 1055.698,A -85,B 0,C 180,E1 -10618.036,E2 -10618.036} C_VEL
LIN {X 0,Y 409.958,Z 1056.449,A -85,B 0,C 180,E1 -10619.018,E2 -10619.018} C_VEL
LIN {X 0,Y 409.946,Z 1056.694,A -85,B 0,C 180,E1 -10620,E2 -10620} C_VEL
LIN {X 0,Y 409.957,Z 1056.335,A -85,B 0,C 180,E1 -10620.983,E2 -10620.983} C_VEL
LIN {X 0,Y 410.024,Z 1055.435,A -85,B 0,C 180,E1 -10621.965,E2 -10621.965} C_VEL
LIN {X 0,Y 410.088,Z 1054.03,A -85,B 0,C 180,E1 -10622.948,E2 -10622.948} C_VEL
LIN {X 0,Y 410.143,Z 1050.895,A -85,B 0,C 180,E1 -10624.423,E2 -10624.423} C_VEL
LIN {X 0,Y 410.406,Z 1046.42,A -85,B 0,C 180,E1 -10625.898,E2 -10625.898} C_VEL
LIN {X 0,Y 410.604,Z 1041.406,A -85,B 0,C 180,E1 -10627.129,E2 -10627.129} C_VEL
LIN {X 0,Y 410.879,Z 1035.038,A -85,B 0,C 180,E1 -10628.36,E2 -10628.36} C_VEL
LIN {X 0,Y 411.226,Z 1028.806,A -85,B 0,C 180,E1 -10629.344,E2 -10629.344} C_VEL
LIN {X 0,Y 411.565,Z 1022.265,A -85,B 0,C 180,E1 -10630.205,E2 -10630.205} C_VEL
LIN {X 0,Y 412,Z 1014.361,A -85,B 0,C 180,E1 -10631.065,E2 -10631.065} C_VEL
LIN {X 0,Y 412.342,Z 1006.04,A -85,B 0,C 180,E1 -10631.802,E2 -10631.802} C_VEL
LIN {X 0,Y 412.741,Z 995.506,A -85,B 0,C 180,E1 -10632.539,E2 -10632.539} C_VEL
LIN {X 0,Y 413.052,Z 984.346,A -85,B 0,C 180,E1 -10633.092,E2 -10633.092} C_VEL
LIN {X 0,Y 413.342,Z 974.335,A -85,B 0,C 180,E1 -10633.427,E2 -10633.427} C_VEL
LIN {X 0,Y 414.079,Z 913.903,A -85,B 0,C 180,E1 -10634.661,E2 -10634.661} C_VEL
LIN {X 0,Y 411.327,Z 898.026,A -85,B 0,C 180,E1 -10635.104,E2 -10635.104} C_VEL
LIN {X 0,Y 411.691,Z 888.456,A -85,B 0,C 180,E1 -10637.896,E2 -10637.896} C_VEL
LIN {X 0,Y 411.303,Z 884.064,A -85,B 0,C 180,E1 -10639.269,E2 -10639.269} C_VEL
LIN {X 0,Y 411.176,Z 884.082,A -85,B 0,C 180,E1 -10643.15,E2 -10643.15} C_VEL
LIN {X 0,Y 411.164,Z 884.077,A -85,B 0,C 180,E1 -10646.387,E2 -10646.387} C_VEL
LIN {X 0,Y 411.193,Z 884.077,A -85,B 0,C 180,E1 -10649.714,E2 -10649.714} C_VEL
LIN {X 0,Y 411.206,Z 884.075,A -85,B 0,C 180,E1 -10653.157,E2 -10653.157} C_VEL
LIN {X 0,Y 411.19,Z 884.074,A -85,B 0,C 180,E1 -10656.552,E2 -10656.552} C_VEL
LIN {X 0,Y 411.168,Z 884.082,A -85,B 0,C 180,E1 -10659.72,E2 -10659.72} C_VEL
LIN {X 0,Y 411.162,Z 884.078,A -85,B 0,C 180,E1 -10663.136,E2 -10663.136} C_VEL
LIN {X 0,Y 411.165,Z 884.081,A -85,B 0,C 180,E1 -10665.882,E2 -10665.882} C_VEL
LIN {X 0,Y 411.158,Z 884.078,A -85,B 0,C 180,E1 -10669.493,E2 -10669.493} C_VEL
LIN {X 0,Y 411.18,Z 884.078,A -85,B 0,C 180,E1 -10672.025,E2 -10672.025} C_VEL
LIN {X 0,Y 411.204,Z 884.073,A -85,B 0,C 180,E1 -10675.124,E2 -10675.124} C_VEL
LIN {X 0,Y 411.162,Z 884.078,A -85,B 0,C 180,E1 -10678.003,E2 -10678.003} C_VEL
LIN {X 0,Y 411.17,Z 884.077,A -85,B 0,C 180,E1 -10681.406,E2 -10681.406} C_VEL
LIN {X 0,Y 411.191,Z 884.081,A -85,B 0,C 180,E1 -10684.942,E2 -10684.942} C_VEL
LIN {X 0,Y 411.203,Z 884.072,A -85,B 0,C 180,E1 -10687.913,E2 -10687.913} C_VEL
LIN {X 0,Y 411.194,Z 884.078,A -85,B 0,C 180,E1 -10691.05,E2 -10691.05} C_VEL
LIN {X 0,Y 411.245,Z 884.067,A -85,B 0,C 180,E1 -10694.131,E2 -10694.131} C_VEL
LIN {X 0,Y 411.306,Z 884.063,A -85,B 0,C 180,E1 -10697.166,E2 -10697.166} C_VEL
LIN {X 0,Y 411.275,Z 884.065,A -85,B 0,C 180,E1 -10700.161,E2 -10700.161} C_VEL
LIN {X 0,Y 411.395,Z 884.049,A -85,B 0,C 180,E1 -10703.132,E2 -10703.132} C_VEL
LIN {X 0,Y 411.285,Z 884.062,A -85,B 0,C 180,E1 -10705.099,E2 -10705.099} C_VEL
LIN {X 0,Y 411.501,Z 884.042,A -85,B 0,C 180,E1 -10708.043,E2 -10708.043} C_VEL
LIN {X 0,Y 411.38,Z 884.05,A -85,B 0,C 180,E1 -10710.979,E2 -10710.979} C_VEL
LIN {X 0,Y 411.415,Z 884.046,A -85,B 0,C 180,E1 -10712.938,E2 -10712.938} C_VEL
LIN {X 0,Y 411.42,Z 884.047,A -85,B 0,C 180,E1 -10715.883,E2 -10715.883} C_VEL
LIN {X 0,Y 411.391,Z 884.05,A -85,B 0,C 180,E1 -10716.948,E2 -10716.948} C_VEL
LIN {X 0,Y 410.702,Z 884.137,A -85,B 0,C 180,E1 -10717.764,E2 -10717.764} C_VEL
LIN {X 0,Y 407.809,Z 884.496,A -85,B 0,C 180,E1 -10719.09,E2 -10719.09} C_VEL
LIN {X 0,Y 405.368,Z 884.802,A -85,B 0,C 180,E1 -10720.161,E2 -10720.161} C_VEL
LIN {X 0,Y 404.317,Z 884.933,A -85,B 0,C 180,E1 -10720.989,E2 -10720.989} C_VEL
LIN {X 0,Y 404.229,Z 884.941,A -85,B 0,C 180,E1 -10721.27,E2 -10721.27} C_VEL
LIN {X 0,Y 404.273,Z 884.937,A -85,B 0,C 180,E1 -10723.211,E2 -10723.211} C_VEL
LIN {X 0,Y 404.181,Z 884.95,A -85,B 0,C 180,E1 -10727.194,E2 -10727.194} C_VEL
LIN {X 0,Y 404.156,Z 884.951,A -85,B 0,C 180,E1 -10730.352,E2 -10730.352} C_VEL
LIN {X 0,Y 404.14,Z 884.954,A -85,B 0,C 180,E1 -10733.577,E2 -10733.577} C_VEL
LIN {X 0,Y 404.135,Z 884.954,A -85,B 0,C 180,E1 -10735.77,E2 -10735.77} C_VEL
LIN {X 0,Y 404.155,Z 884.954,A -85,B 0,C 180,E1 -10739.602,E2 -10739.602} C_VEL
LIN {X 0,Y 404.17,Z 884.954,A -85,B 0,C 180,E1 -10743.419,E2 -10743.419} C_VEL
LIN {X 0,Y 404.136,Z 884.954,A -85,B 0,C 180,E1 -10746.247,E2 -10746.247} C_VEL
LIN {X 0,Y 404.135,Z 884.953,A -85,B 0,C 180,E1 -10748.76,E2 -10748.76} C_VEL
LIN {X 0,Y 404.108,Z 884.959,A -85,B 0,C 180,E1 -10751.596,E2 -10751.596} C_VEL
LIN {X 0,Y 404.146,Z 884.953,A -85,B 0,C 180,E1 -10754.521,E2 -10754.521} C_VEL
LIN {X 0,Y 404.124,Z 884.954,A -85,B 0,C 180,E1 -10757.293,E2 -10757.293} C_VEL
LIN {X 0,Y 404.137,Z 884.956,A -85,B 0,C 180,E1 -10759.951,E2 -10759.951} C_VEL
LIN {X 0,Y 404.133,Z 884.953,A -85,B 0,C 180,E1 -10763.126,E2 -10763.126} C_VEL
LIN {X 0,Y 404.141,Z 884.955,A -85,B 0,C 180,E1 -10766.187,E2 -10766.187} C_VEL
LIN {X 0,Y 404.143,Z 884.952,A -85,B 0,C 180,E1 -10769.714,E2 -10769.714} C_VEL
LIN {X 0,Y 404.1,Z 884.961,A -85,B 0,C 180,E1 -10773.115,E2 -10773.115} C_VEL
LIN {X 0,Y 404.132,Z 884.956,A -85,B 0,C 180,E1 -10775.331,E2 -10775.331} C_VEL
LIN {X 0,Y 404.134,Z 884.954,A -85,B 0,C 180,E1 -10778.58,E2 -10778.58} C_VEL
LIN {X 0,Y 404.156,Z 884.951,A -85,B 0,C 180,E1 -10781.759,E2 -10781.759} C_VEL
LIN {X 0,Y 404.162,Z 884.951,A -85,B 0,C 180,E1 -10784.88,E2 -10784.88} C_VEL
LIN {X 0,Y 404.248,Z 884.941,A -85,B 0,C 180,E1 -10787.958,E2 -10787.958} C_VEL
LIN {X 0,Y 404.345,Z 884.93,A -85,B 0,C 180,E1 -10792.007,E2 -10792.007} C_VEL
LIN {X 0,Y 404.369,Z 884.928,A -85,B 0,C 180,E1 -10794.014,E2 -10794.014} C_VEL
LIN {X 0,Y 404.468,Z 884.918,A -85,B 0,C 180,E1 -10798.008,E2 -10798.008} C_VEL
LIN {X 0,Y 404.349,Z 884.926,A -85,B 0,C 180,E1 -10800.995,E2 -10800.995} C_VEL
LIN {X 0,Y 404.348,Z 884.926,A -85,B 0,C 180,E1 -10802.988,E2 -10802.988} C_VEL
LIN {X 0,Y 404.368,Z 884.927,A -85,B 0,C 180,E1 -10805.985,E2 -10805.985} C_VEL
LIN {X 0,Y 404.256,Z 884.939,A -85,B 0,C 180,E1 -10809.001,E2 -10809.001} C_VEL
LIN {X 0,Y 404.247,Z 884.94,A -85,B 0,C 180,E1 -10812.041,E2 -10812.041} C_VEL
LIN {X 0,Y 404.161,Z 884.952,A -85,B 0,C 180,E1 -10815.119,E2 -10815.119} C_VEL
LIN {X 0,Y 404.154,Z 884.951,A -85,B 0,C 180,E1 -10818.24,E2 -10818.24} C_VEL
LIN {X 0,Y 404.131,Z 884.955,A -85,B 0,C 180,E1 -10821.419,E2 -10821.419} C_VEL
LIN {X 0,Y 404.128,Z 884.955,A -85,B 0,C 180,E1 -10824.668,E2 -10824.668} C_VEL
LIN {X 0,Y 404.099,Z 884.957,A -85,B 0,C 180,E1 -10828.006,E2 -10828.006} C_VEL
LIN {X 0,Y 404.139,Z 884.952,A -85,B 0,C 180,E1 -10830.285,E2 -10830.285} C_VEL
LIN {X 0,Y 404.136,Z 884.956,A -85,B 0,C 180,E1 -10833.813,E2 -10833.813} C_VEL
LIN {X 0,Y 404.129,Z 884.954,A -85,B 0,C 180,E1 -10836.873,E2 -10836.873} C_VEL
LIN {X 0,Y 404.117,Z 884.959,A -85,B 0,C 180,E1 -10840.074,E2 -10840.074} C_VEL
LIN {X 0,Y 404.14,Z 884.952,A -85,B 0,C 180,E1 -10843.081,E2 -10843.081} C_VEL
LIN {X 0,Y 404.119,Z 884.96,A -85,B 0,C 180,E1 -10845.922,E2 -10845.922} C_VEL
LIN {X 0,Y 404.099,Z 884.959,A -85,B 0,C 180,E1 -10848.632,E2 -10848.632} C_VEL
LIN {X 0,Y 404.132,Z 884.953,A -85,B 0,C 180,E1 -10851.496,E2 -10851.496} C_VEL
LIN {X 0,Y 404.175,Z 884.949,A -85,B 0,C 180,E1 -10854.983,E2 -10854.983} C_VEL
LIN {X 0,Y 404.132,Z 884.958,A -85,B 0,C 180,E1 -10858.443,E2 -10858.443} C_VEL
LIN {X 0,Y 404.145,Z 884.957,A -85,B 0,C 180,E1 -10860.862,E2 -10860.862} C_VEL
LIN {X 0,Y 404.188,Z 885.06,A -85,B 0,C 180,E1 -10864.095,E2 -10864.095} C_VEL
LIN {X 0,Y 406.172,Z 895.873,A -85,B 0,C 180,E1 -10866.826,E2 -10866.826} C_VEL
LIN {X 0,Y 405.884,Z 903.657,A -85,B 0,C 180,E1 -10868.677,E2 -10868.677} C_VEL
LIN {X 0,Y 404.91,Z 919.463,A -85,B 0,C 180,E1 -10872.369,E2 -10872.369} C_VEL
LIN {X 0,Y 404.326,Z 929.381,A -85,B 0,C 180,E1 -10874.661,E2 -10874.661} C_VEL
LIN {X 0,Y 407.061,Z 952.44,A -85,B 0,C 180,E1 -10875.26,E2 -10875.26} C_VEL
LIN {X 0,Y 406.341,Z 1007.755,A -85,B 0,C 180,E1 -10876.433,E2 -10876.433} C_VEL
LIN {X 0,Y 405.882,Z 1019.699,A -85,B 0,C 180,E1 -10876.864,E2 -10876.864} C_VEL
LIN {X 0,Y 405.448,Z 1030.771,A -85,B 0,C 180,E1 -10877.486,E2 -10877.486} C_VEL
LIN {X 0,Y 405.046,Z 1039.28,A -85,B 0,C 180,E1 -10878.109,E2 -10878.109} C_VEL
LIN {X 0,Y 404.644,Z 1047.502,A -85,B 0,C 180,E1 -10878.859,E2 -10878.859} C_VEL
LIN {X 0,Y 404.186,Z 1055.33,A -85,B 0,C 180,E1 -10879.733,E2 -10879.733} C_VEL
LIN {X 0,Y 403.725,Z 1064.36,A -85,B 0,C 180,E1 -10880.986,E2 -10880.986} C_VEL
LIN {X 0,Y 403.411,Z 1071.321,A -85,B 0,C 180,E1 -10882.24,E2 -10882.24} C_VEL
LIN {X 0,Y 403.223,Z 1075.986,A -85,B 0,C 180,E1 -10883.266,E2 -10883.266} C_VEL
LIN {X 0,Y 403.034,Z 1080.468,A -85,B 0,C 180,E1 -10884.496,E2 -10884.496} C_VEL
LIN {X 0,Y 402.912,Z 1084.576,A -85,B 0,C 180,E1 -10885.999,E2 -10885.999} C_VEL
LIN {X 0,Y 402.889,Z 1086.541,A -85,B 0,C 180,E1 -10887,E2 -10887} C_VEL
LIN {X 0,Y 402.933,Z 1087.967,A -85,B 0,C 180,E1 -10888.001,E2 -10888.001} C_VEL
LIN {X 0,Y 402.879,Z 1088.866,A -85,B 0,C 180,E1 -10889,E2 -10889} C_VEL
LIN {X 0,Y 402.868,Z 1089.169,A -85,B 0,C 180,E1 -10890,E2 -10890} C_VEL
LIN {X 0,Y 402.879,Z 1088.899,A -85,B 0,C 180,E1 -10890.999,E2 -10890.999} C_VEL
LIN {X 0,Y 402.914,Z 1088.126,A -85,B 0,C 180,E1 -10891.999,E2 -10891.999} C_VEL
LIN {X 0,Y 402.88,Z 1086.838,A -85,B 0,C 180,E1 -10893,E2 -10893} C_VEL
LIN {X 0,Y 402.972,Z 1083.8,A -85,B 0,C 180,E1 -10894.501,E2 -10894.501} C_VEL
LIN {X 0,Y 403.034,Z 1081.036,A -85,B 0,C 180,E1 -10895.503,E2 -10895.503} C_VEL
LIN {X 0,Y 403.279,Z 1075.606,A -85,B 0,C 180,E1 -10897.007,E2 -10897.007} C_VEL
LIN {X 0,Y 403.587,Z 1068.442,A -85,B 0,C 180,E1 -10898.512,E2 -10898.512} C_VEL
LIN {X 0,Y 404.058,Z 1060.636,A -85,B 0,C 180,E1 -10899.764,E2 -10899.764} C_VEL
LIN {X 0,Y 404.476,Z 1054.024,A -85,B 0,C 180,E1 -10900.639,E2 -10900.639} C_VEL
LIN {X 0,Y 404.941,Z 1046.052,A -85,B 0,C 180,E1 -10901.513,E2 -10901.513} C_VEL
LIN {X 0,Y 405.412,Z 1037.688,A -85,B 0,C 180,E1 -10902.26,E2 -10902.26} C_VEL
LIN {X 0,Y 405.91,Z 1027.143,A -85,B 0,C 180,E1 -10903.008,E2 -10903.008} C_VEL
LIN {X 0,Y 406.45,Z 1016.056,A -85,B 0,C 180,E1 -10903.563,E2 -10903.563} C_VEL
LIN {X 0,Y 406.84,Z 1006.285,A -85,B 0,C 180,E1 -10903.9,E2 -10903.9} C_VEL
LIN {X 0,Y 407.584,Z 950.689,A -85,B 0,C 180,E1 -10905.146,E2 -10905.146} C_VEL
LIN {X 0,Y 405.527,Z 933.684,A -85,B 0,C 180,E1 -10905.657,E2 -10905.657} C_VEL
LIN {X 0,Y 404.529,Z 927.799,A -85,B 0,C 180,E1 -10905.854,E2 -10905.854} C_VEL
LIN {X 0,Y 405.504,Z 912.566,A -85,B 0,C 180,E1 -10909.489,E2 -10909.489} C_VEL
LIN {X 0,Y 406.415,Z 900.936,A -85,B 0,C 180,E1 -10912.361,E2 -10912.361} C_VEL
LIN {X 0,Y 406.538,Z 897.821,A -85,B 0,C 180,E1 -10913.159,E2 -10913.159} C_VEL
LIN {X 0,Y 404.993,Z 888.763,A -85,B 0,C 180,E1 -10915.711,E2 -10915.711} C_VEL
LIN {X 0,Y 404.131,Z 884.962,A -85,B 0,C 180,E1 -10916.882,E2 -10916.882} C_VEL
LIN {X 0,Y 404.137,Z 884.957,A -85,B 0,C 180,E1 -10920.286,E2 -10920.286} C_VEL
LIN {X 0,Y 404.135,Z 884.959,A -85,B 0,C 180,E1 -10923.813,E2 -10923.813} C_VEL
LIN {X 0,Y 404.127,Z 884.957,A -85,B 0,C 180,E1 -10926.874,E2 -10926.874} C_VEL
LIN {X 0,Y 404.115,Z 884.959,A -85,B 0,C 180,E1 -10930.075,E2 -10930.075} C_VEL
LIN {X 0,Y 404.138,Z 884.955,A -85,B 0,C 180,E1 -10933.082,E2 -10933.082} C_VEL
LIN {X 0,Y 404.117,Z 884.961,A -85,B 0,C 180,E1 -10935.922,E2 -10935.922} C_VEL
LIN {X 0,Y 404.098,Z 884.96,A -85,B 0,C 180,E1 -10938.633,E2 -10938.633} C_VEL
LIN {X 0,Y 404.131,Z 884.957,A -85,B 0,C 180,E1 -10941.496,E2 -10941.496} C_VEL
LIN {X 0,Y 404.17,Z 884.951,A -85,B 0,C 180,E1 -10944.983,E2 -10944.983} C_VEL
LIN {X 0,Y 404.132,Z 884.959,A -85,B 0,C 180,E1 -10948.444,E2 -10948.444} C_VEL
LIN {X 0,Y 404.145,Z 884.958,A -85,B 0,C 180,E1 -10950.862,E2 -10950.862} C_VEL
LIN {X 0,Y 404.15,Z 884.959,A -85,B 0,C 180,E1 -10954.724,E2 -10954.724} C_VEL
LIN {X 0,Y 404.162,Z 884.959,A -85,B 0,C 180,E1 -10957.508,E2 -10957.508} C_VEL
LIN {X 0,Y 404.16,Z 885.055,A -85,B 0,C 180,E1 -10958.983,E2 -10958.983} C_VEL
LIN {X 0,Y 405.293,Z 891.409,A -85,B 0,C 180,E1 -10961.289,E2 -10961.289} C_VEL
LIN {X 0,Y 405.149,Z 897.68,A -85,B 0,C 180,E1 -10963.369,E2 -10963.369} C_VEL
LIN {X 0,Y 404.969,Z 900.633,A -85,B 0,C 180,E1 -10964.251,E2 -10964.251} C_VEL
LIN {X 0,Y 407.847,Z 913.719,A -85,B 0,C 180,E1 -10964.725,E2 -10964.725} C_VEL
LIN {X 0,Y 408.096,Z 918.186,A -85,B 0,C 180,E1 -10964.847,E2 -10964.847} C_VEL
LIN {X 0,Y 406.926,Z 977.821,A -85,B 0,C 180,E1 -10966.199,E2 -10966.199} C_VEL
LIN {X 0,Y 406.56,Z 990.088,A -85,B 0,C 180,E1 -10966.696,E2 -10966.696} C_VEL
LIN {X 0,Y 406.112,Z 999.669,A -85,B 0,C 180,E1 -10967.253,E2 -10967.253} C_VEL
LIN {X 0,Y 405.783,Z 1007.975,A -85,B 0,C 180,E1 -10967.878,E2 -10967.878} C_VEL
LIN {X 0,Y 405.386,Z 1016.035,A -85,B 0,C 180,E1 -10968.627,E2 -10968.627} C_VEL
LIN {X 0,Y 404.924,Z 1023.735,A -85,B 0,C 180,E1 -10969.5,E2 -10969.5} C_VEL
LIN {X 0,Y 404.303,Z 1032.602,A -85,B 0,C 180,E1 -10970.748,E2 -10970.748} C_VEL
LIN {X 0,Y 403.885,Z 1039.43,A -85,B 0,C 180,E1 -10971.998,E2 -10971.998} C_VEL
LIN {X 0,Y 403.646,Z 1045.04,A -85,B 0,C 180,E1 -10973.29,E2 -10973.29} C_VEL
LIN {X 0,Y 403.282,Z 1049.207,A -85,B 0,C 180,E1 -10974.5,E2 -10974.5} C_VEL
LIN {X 0,Y 403.197,Z 1051.892,A -85,B 0,C 180,E1 -10975.502,E2 -10975.502} C_VEL
LIN {X 0,Y 403.093,Z 1054.811,A -85,B 0,C 180,E1 -10977.002,E2 -10977.002} C_VEL
LIN {X 0,Y 402.967,Z 1056.04,A -85,B 0,C 180,E1 -10978.001,E2 -10978.001} C_VEL
LIN {X 0,Y 402.885,Z 1056.763,A -85,B 0,C 180,E1 -10979.001,E2 -10979.001} C_VEL
LIN {X 0,Y 402.87,Z 1056.982,A -85,B 0,C 180,E1 -10980,E2 -10980} C_VEL
LIN {X 0,Y 402.884,Z 1056.609,A -85,B 0,C 180,E1 -10981,E2 -10981} C_VEL
LIN {X 0,Y 402.956,Z 1055.672,A -85,B 0,C 180,E1 -10981.999,E2 -10981.999} C_VEL
LIN {X 0,Y 402.994,Z 1054.228,A -85,B 0,C 180,E1 -10982.999,E2 -10982.999} C_VEL
LIN {X 0,Y 403.067,Z 1051.038,A -85,B 0,C 180,E1 -10984.501,E2 -10984.501} C_VEL
LIN {X 0,Y 403.334,Z 1046.476,A -85,B 0,C 180,E1 -10986.002,E2 -10986.002} C_VEL
LIN {X 0,Y 403.56,Z 1041.371,A -85,B 0,C 180,E1 -10987.254,E2 -10987.254} C_VEL
LIN {X 0,Y 403.841,Z 1034.924,A -85,B 0,C 180,E1 -10988.507,E2 -10988.507} C_VEL
LIN {X 0,Y 404.198,Z 1028.604,A -85,B 0,C 180,E1 -10989.508,E2 -10989.508} C_VEL
LIN {X 0,Y 404.652,Z 1020.926,A -85,B 0,C 180,E1 -10990.508,E2 -10990.508} C_VEL
LIN {X 0,Y 405.148,Z 1011.424,A -85,B 0,C 180,E1 -10991.508,E2 -10991.508} C_VEL
LIN {X 0,Y 405.573,Z 1002.22,A -85,B 0,C 180,E1 -10992.256,E2 -10992.256} C_VEL
LIN {X 0,Y 405.88,Z 992.223,A -85,B 0,C 180,E1 -10992.882,E2 -10992.882} C_VEL
LIN {X 0,Y 406.089,Z 982.865,A -85,B 0,C 180,E1 -10993.321,E2 -10993.321} C_VEL
LIN {X 0,Y 406.389,Z 973.271,A -85,B 0,C 180,E1 -10993.629,E2 -10993.629} C_VEL
LIN {X 0,Y 407.084,Z 914.35,A -85,B 0,C 180,E1 -10994.867,E2 -10994.867} C_VEL
LIN {X 0,Y 404.322,Z 898.331,A -85,B 0,C 180,E1 -10995.308,E2 -10995.308} C_VEL
LIN {X 0,Y 404.673,Z 890.238,A -85,B 0,C 180,E1 -10997.693,E2 -10997.693} C_VEL
LIN {X 0,Y 404.245,Z 884.943,A -85,B 0,C 180,E1 -10999.345,E2 -10999.345} C_VEL
LIN {X 0,Y 404.141,Z 884.956,A -85,B 0,C 180,E1 -11002.829,E2 -11002.829} C_VEL
LIN {X 0,Y 404.132,Z 884.954,A -85,B 0,C 180,E1 -11005.771,E2 -11005.771} C_VEL
LIN {X 0,Y 404.152,Z 884.955,A -85,B 0,C 180,E1 -11009.602,E2 -11009.602} C_VEL
LIN {X 0,Y 404.139,Z 884.952,A -85,B 0,C 180,E1 -11012.623,E2 -11012.623} C_VEL
LIN {X 0,Y 404.151,Z 884.953,A -85,B 0,C 180,E1 -11015.184,E2 -11015.184} C_VEL
LIN {X 0,Y 404.133,Z 884.953,A -85,B 0,C 180,E1 -11018.76,E2 -11018.76} C_VEL
LIN {X 0,Y 404.106,Z 884.96,A -85,B 0,C 180,E1 -11021.597,E2 -11021.597} C_VEL
LIN {X 0,Y 404.144,Z 884.953,A -85,B 0,C 180,E1 -11024.522,E2 -11024.522} C_VEL
LIN {X 0,Y 404.122,Z 884.955,A -85,B 0,C 180,E1 -11027.294,E2 -11027.294} C_VEL
LIN {X 0,Y 404.135,Z 884.956,A -85,B 0,C 180,E1 -11029.951,E2 -11029.951} C_VEL
LIN {X 0,Y 404.133,Z 884.953,A -85,B 0,C 180,E1 -11033.127,E2 -11033.127} C_VEL
LIN {X 0,Y 404.14,Z 884.955,A -85,B 0,C 180,E1 -11036.187,E2 -11036.187} C_VEL
LIN {X 0,Y 404.142,Z 884.952,A -85,B 0,C 180,E1 -11039.715,E2 -11039.715} C_VEL
LIN {X 0,Y 404.1,Z 884.961,A -85,B 0,C 180,E1 -11043.116,E2 -11043.116} C_VEL
LIN {X 0,Y 404.15,Z 884.952,A -85,B 0,C 180,E1 -11046.424,E2 -11046.424} C_VEL
LIN {X 0,Y 404.154,Z 884.951,A -85,B 0,C 180,E1 -11049.891,E2 -11049.891} C_VEL
LIN {X 0,Y 404.22,Z 884.945,A -85,B 0,C 180,E1 -11052.994,E2 -11052.994} C_VEL
LIN {X 0,Y 404.288,Z 884.935,A -85,B 0,C 180,E1 -11056.939,E2 -11056.939} C_VEL
LIN {X 0,Y 404.243,Z 884.942,A -85,B 0,C 180,E1 -11059.988,E2 -11059.988} C_VEL
LIN {X 0,Y 404.345,Z 884.927,A -85,B 0,C 180,E1 -11063.012,E2 -11063.012} C_VEL
LIN {X 0,Y 404.257,Z 884.938,A -85,B 0,C 180,E1 -11065.013,E2 -11065.013} C_VEL
LIN {X 0,Y 404.47,Z 884.918,A -85,B 0,C 180,E1 -11068.009,E2 -11068.009} C_VEL
LIN {X 0,Y 404.351,Z 884.926,A -85,B 0,C 180,E1 -11070.996,E2 -11070.996} C_VEL
LIN {X 0,Y 404.35,Z 884.926,A -85,B 0,C 180,E1 -11072.989,E2 -11072.989} C_VEL
LIN {X 0,Y 404.371,Z 884.926,A -85,B 0,C 180,E1 -11075.986,E2 -11075.986} C_VEL
LIN {X 0,Y 404.259,Z 884.939,A -85,B 0,C 180,E1 -11079.002,E2 -11079.002} C_VEL
LIN {X 0,Y 404.229,Z 884.941,A -85,B 0,C 180,E1 -11081.27,E2 -11081.27} C_VEL
LIN {X 0,Y 403.552,Z 885.029,A -85,B 0,C 180,E1 -11082.101,E2 -11082.101} C_VEL
LIN {X 0,Y 400.674,Z 885.384,A -85,B 0,C 180,E1 -11083.452,E2 -11083.452} C_VEL
LIN {X 0,Y 398.239,Z 885.692,A -85,B 0,C 180,E1 -11084.543,E2 -11084.543} C_VEL
LIN {X 0,Y 397.192,Z 885.818,A -85,B 0,C 180,E1 -11085.387,E2 -11085.387} C_VEL
LIN {X 0,Y 397.105,Z 885.828,A -85,B 0,C 180,E1 -11085.672,E2 -11085.672} C_VEL
LIN {X 0,Y 397.104,Z 885.832,A -85,B 0,C 180,E1 -11088.577,E2 -11088.577} C_VEL
LIN {X 0,Y 397.094,Z 885.83,A -85,B 0,C 180,E1 -11091.819,E2 -11091.819} C_VEL
LIN {X 0,Y 397.104,Z 885.835,A -85,B 0,C 180,E1 -11095.135,E2 -11095.135} C_VEL
LIN {X 0,Y 397.064,Z 885.834,A -85,B 0,C 180,E1 -11098.548,E2 -11098.548} C_VEL
LIN {X 0,Y 397.079,Z 885.834,A -85,B 0,C 180,E1 -11101.834,E2 -11101.834} C_VEL
LIN {X 0,Y 397.119,Z 885.827,A -85,B 0,C 180,E1 -11104.494,E2 -11104.494} C_VEL
LIN {X 0,Y 397.092,Z 885.831,A -85,B 0,C 180,E1 -11108.277,E2 -11108.277} C_VEL
LIN {X 0,Y 397.054,Z 885.841,A -85,B 0,C 180,E1 -11111.976,E2 -11111.976} C_VEL
LIN {X 0,Y 397.088,Z 885.83,A -85,B 0,C 180,E1 -11115.069,E2 -11115.069} C_VEL
LIN {X 0,Y 397.054,Z 885.84,A -85,B 0,C 180,E1 -11118.024,E2 -11118.024} C_VEL
LIN {X 0,Y 397.089,Z 885.831,A -85,B 0,C 180,E1 -11121.723,E2 -11121.723} C_VEL
LIN {X 0,Y 397.122,Z 885.826,A -85,B 0,C 180,E1 -11125.506,E2 -11125.506} C_VEL
LIN {X 0,Y 397.076,Z 885.834,A -85,B 0,C 180,E1 -11129.117,E2 -11129.117} C_VEL
LIN {X 0,Y 397.061,Z 885.835,A -85,B 0,C 180,E1 -11132.253,E2 -11132.253} C_VEL
LIN {X 0,Y 397.104,Z 885.835,A -85,B 0,C 180,E1 -11134.864,E2 -11134.864} C_VEL
LIN {X 0,Y 397.094,Z 885.83,A -85,B 0,C 180,E1 -11138.181,E2 -11138.181} C_VEL
LIN {X 0,Y 397.103,Z 885.833,A -85,B 0,C 180,E1 -11141.423,E2 -11141.423} C_VEL
LIN {X 0,Y 397.126,Z 885.83,A -85,B 0,C 180,E1 -11143.551,E2 -11143.551} C_VEL
LIN {X 0,Y 397.233,Z 885.813,A -85,B 0,C 180,E1 -11146.702,E2 -11146.702} C_VEL
LIN {X 0,Y 397.203,Z 885.82,A -85,B 0,C 180,E1 -11149.808,E2 -11149.808} C_VEL
LIN {X 0,Y 397.296,Z 885.805,A -85,B 0,C 180,E1 -11152.886,E2 -11152.886} C_VEL
LIN {X 0,Y 397.226,Z 885.813,A -85,B 0,C 180,E1 -11154.924,E2 -11154.924} C_VEL
LIN {X 0,Y 397.435,Z 885.794,A -85,B 0,C 180,E1 -11157.973,E2 -11157.973} C_VEL
LIN {X 0,Y 397.32,Z 885.802,A -85,B 0,C 180,E1 -11161.013,E2 -11161.013} C_VEL
LIN {X 0,Y 397.284,Z 885.806,A -85,B 0,C 180,E1 -11163.042,E2 -11163.042} C_VEL
LIN {X 0,Y 397.321,Z 885.806,A -85,B 0,C 180,E1 -11166.092,E2 -11166.092} C_VEL
LIN {X 0,Y 397.227,Z 885.813,A -85,B 0,C 180,E1 -11169.162,E2 -11169.162} C_VEL
LIN {X 0,Y 397.213,Z 885.818,A -85,B 0,C 180,E1 -11172.258,E2 -11172.258} C_VEL
LIN {X 0,Y 397.113,Z 885.828,A -85,B 0,C 180,E1 -11175.394,E2 -11175.394} C_VEL
LIN {X 0,Y 397.121,Z 885.827,A -85,B 0,C 180,E1 -11177.509,E2 -11177.509} C_VEL
LIN {X 0,Y 397.095,Z 885.834,A -85,B 0,C 180,E1 -11180.73,E2 -11180.73} C_VEL
LIN {X 0,Y 397.097,Z 885.829,A -85,B 0,C 180,E1 -11184.02,E2 -11184.02} C_VEL
LIN {X 0,Y 397.062,Z 885.839,A -85,B 0,C 180,E1 -11187.4,E2 -11187.4} C_VEL
LIN {X 0,Y 397.095,Z 885.831,A -85,B 0,C 180,E1 -11189.861,E2 -11189.861} C_VEL
LIN {X 0,Y 397.11,Z 885.832,A -85,B 0,C 180,E1 -11193.273,E2 -11193.273} C_VEL
LIN {X 0,Y 397.091,Z 885.831,A -85,B 0,C 180,E1 -11196.995,E2 -11196.995} C_VEL
LIN {X 0,Y 397.054,Z 885.836,A -85,B 0,C 180,E1 -11200.437,E2 -11200.437} C_VEL
LIN {X 0,Y 397.086,Z 885.834,A -85,B 0,C 180,E1 -11203.65,E2 -11203.65} C_VEL
LIN {X 0,Y 397.09,Z 885.833,A -85,B 0,C 180,E1 -11206.522,E2 -11206.522} C_VEL
LIN {X 0,Y 397.083,Z 885.836,A -85,B 0,C 180,E1 -11210.419,E2 -11210.419} C_VEL
LIN {X 0,Y 397.091,Z 885.831,A -85,B 0,C 180,E1 -11213.004,E2 -11213.004} C_VEL
LIN {X 0,Y 397.097,Z 885.833,A -85,B 0,C 180,E1 -11216.286,E2 -11216.286} C_VEL
LIN {X 0,Y 397.071,Z 885.835,A -85,B 0,C 180,E1 -11219.117,E2 -11219.117} C_VEL
LIN {X 0,Y 397.056,Z 885.836,A -85,B 0,C 180,E1 -11222.253,E2 -11222.253} C_VEL
LIN {X 0,Y 397.152,Z 885.933,A -85,B 0,C 180,E1 -11223.934,E2 -11223.934} C_VEL
LIN {X 0,Y 399.19,Z 897.089,A -85,B 0,C 180,E1 -11226.799,E2 -11226.799} C_VEL
LIN {X 0,Y 398.678,Z 907.701,A -85,B 0,C 180,E1 -11229.355,E2 -11229.355} C_VEL
LIN {X 0,Y 397.712,Z 921.902,A -85,B 0,C 180,E1 -11232.726,E2 -11232.726} C_VEL
LIN {X 0,Y 397.326,Z 929.223,A -85,B 0,C 180,E1 -11234.449,E2 -11234.449} C_VEL
LIN {X 0,Y 400.104,Z 953.266,A -85,B 0,C 180,E1 -11235.08,E2 -11235.08} C_VEL
LIN {X 0,Y 399.372,Z 1007.261,A -85,B 0,C 180,E1 -11236.257,E2 -11236.257} C_VEL
LIN {X 0,Y 398.888,Z 1019.26,A -85,B 0,C 180,E1 -11236.694,E2 -11236.694} C_VEL
LIN {X 0,Y 398.503,Z 1029.448,A -85,B 0,C 180,E1 -11237.264,E2 -11237.264} C_VEL
LIN {X 0,Y 398.091,Z 1038.154,A -85,B 0,C 180,E1 -11237.898,E2 -11237.898} C_VEL
LIN {X 0,Y 397.633,Z 1046.52,A -85,B 0,C 180,E1 -11238.66,E2 -11238.66} C_VEL
LIN {X 0,Y 397.195,Z 1054.472,A -85,B 0,C 180,E1 -11239.551,E2 -11239.551} C_VEL
LIN {X 0,Y 396.78,Z 1061.927,A -85,B 0,C 180,E1 -11240.57,E2 -11240.57} C_VEL
LIN {X 0,Y 396.382,Z 1069.478,A -85,B 0,C 180,E1 -11241.845,E2 -11241.845} C_VEL
LIN {X 0,Y 396.152,Z 1075.697,A -85,B 0,C 180,E1 -11243.211,E2 -11243.211} C_VEL
LIN {X 0,Y 395.938,Z 1079.984,A -85,B 0,C 180,E1 -11244.397,E2 -11244.397} C_VEL
LIN {X 0,Y 395.837,Z 1084.148,A -85,B 0,C 180,E1 -11245.927,E2 -11245.927} C_VEL
LIN {X 0,Y 395.792,Z 1086.156,A -85,B 0,C 180,E1 -11246.946,E2 -11246.946} C_VEL
LIN {X 0,Y 395.846,Z 1087.622,A -85,B 0,C 180,E1 -11247.965,E2 -11247.965} C_VEL
LIN {X 0,Y 395.808,Z 1088.548,A -85,B 0,C 180,E1 -11248.982,E2 -11248.982} C_VEL
LIN {X 0,Y 395.794,Z 1088.859,A -85,B 0,C 180,E1 -11250,E2 -11250} C_VEL
LIN {X 0,Y 395.808,Z 1088.617,A -85,B 0,C 180,E1 -11251.017,E2 -11251.017} C_VEL
LIN {X 0,Y 395.813,Z 1087.87,A -85,B 0,C 180,E1 -11252.035,E2 -11252.035} C_VEL
LIN {X 0,Y 395.781,Z 1086.604,A -85,B 0,C 180,E1 -11253.054,E2 -11253.054} C_VEL
LIN {X 0,Y 395.836,Z 1084.794,A -85,B 0,C 180,E1 -11254.072,E2 -11254.072} C_VEL
LIN {X 0,Y 395.938,Z 1080.827,A -85,B 0,C 180,E1 -11255.602,E2 -11255.602} C_VEL
LIN {X 0,Y 396.151,Z 1076.788,A -85,B 0,C 180,E1 -11256.789,E2 -11256.789} C_VEL
LIN {X 0,Y 396.417,Z 1070.879,A -85,B 0,C 180,E1 -11258.154,E2 -11258.154} C_VEL
LIN {X 0,Y 396.86,Z 1063.943,A -85,B 0,C 180,E1 -11259.428,E2 -11259.428} C_VEL
LIN {X 0,Y 397.436,Z 1055.095,A -85,B 0,C 180,E1 -11260.7,E2 -11260.7} C_VEL
LIN {X 0,Y 397.913,Z 1047.38,A -85,B 0,C 180,E1 -11261.59,E2 -11261.59} C_VEL
LIN {X 0,Y 398.403,Z 1039.347,A -85,B 0,C 180,E1 -11262.35,E2 -11262.35} C_VEL
LIN {X 0,Y 398.802,Z 1031.14,A -85,B 0,C 180,E1 -11262.985,E2 -11262.985} C_VEL
LIN {X 0,Y 399.274,Z 1021.785,A -85,B 0,C 180,E1 -11263.552,E2 -11263.552} C_VEL
LIN {X 0,Y 399.87,Z 1010.474,A -85,B 0,C 180,E1 -11264.05,E2 -11264.05} C_VEL
LIN {X 0,Y 400.285,Z 993.972,A -85,B 0,C 180,E1 -11264.478,E2 -11264.478} C_VEL
LIN {X 0,Y 400.877,Z 951.621,A -85,B 0,C 180,E1 -11265.454,E2 -11265.454} C_VEL
LIN {X 0,Y 398.894,Z 934.89,A -85,B 0,C 180,E1 -11265.976,E2 -11265.976} C_VEL
LIN {X 0,Y 397.597,Z 927.401,A -85,B 0,C 180,E1 -11266.247,E2 -11266.247} C_VEL
LIN {X 0,Y 398.708,Z 911.654,A -85,B 0,C 180,E1 -11270.104,E2 -11270.104} C_VEL
LIN {X 0,Y 399.638,Z 901.205,A -85,B 0,C 180,E1 -11272.761,E2 -11272.761} C_VEL
LIN {X 0,Y 399.327,Z 897.141,A -85,B 0,C 180,E1 -11273.878,E2 -11273.878} C_VEL
LIN {X 0,Y 397.858,Z 889.276,A -85,B 0,C 180,E1 -11276.207,E2 -11276.207} C_VEL
LIN {X 0,Y 397.065,Z 885.841,A -85,B 0,C 180,E1 -11277.328,E2 -11277.328} C_VEL
LIN {X 0,Y 397.092,Z 885.835,A -85,B 0,C 180,E1 -11279.862,E2 -11279.862} C_VEL
LIN {X 0,Y 397.109,Z 885.835,A -85,B 0,C 180,E1 -11283.273,E2 -11283.273} C_VEL
LIN {X 0,Y 397.089,Z 885.834,A -85,B 0,C 180,E1 -11286.996,E2 -11286.996} C_VEL
LIN {X 0,Y 397.052,Z 885.837,A -85,B 0,C 180,E1 -11290.437,E2 -11290.437} C_VEL
LIN {X 0,Y 397.084,Z 885.836,A -85,B 0,C 180,E1 -11293.651,E2 -11293.651} C_VEL
LIN {X 0,Y 397.088,Z 885.833,A -85,B 0,C 180,E1 -11296.523,E2 -11296.523} C_VEL
LIN {X 0,Y 397.082,Z 885.835,A -85,B 0,C 180,E1 -11300.419,E2 -11300.419} C_VEL
LIN {X 0,Y 397.089,Z 885.833,A -85,B 0,C 180,E1 -11303.004,E2 -11303.004} C_VEL
LIN {X 0,Y 397.109,Z 885.833,A -85,B 0,C 180,E1 -11306.727,E2 -11306.727} C_VEL
LIN {X 0,Y 397.111,Z 885.834,A -85,B 0,C 180,E1 -11310.295,E2 -11310.295} C_VEL
LIN {X 0,Y 397.068,Z 885.837,A -85,B 0,C 180,E1 -11313.737,E2 -11313.737} C_VEL
LIN {X 0,Y 397.098,Z 885.84,A -85,B 0,C 180,E1 -11317.085,E2 -11317.085} C_VEL
LIN {X 0,Y 397.124,Z 885.947,A -85,B 0,C 180,E1 -11318.592,E2 -11318.592} C_VEL
LIN {X 0,Y 398.279,Z 892.218,A -85,B 0,C 180,E1 -11320.947,E2 -11320.947} C_VEL
LIN {X 0,Y 398.352,Z 896.851,A -85,B 0,C 180,E1 -11322.547,E2 -11322.547} C_VEL
LIN {X 0,Y 398.108,Z 901.09,A -85,B 0,C 180,E1 -11323.877,E2 -11323.877} C_VEL
LIN {X 0,Y 401.286,Z 915.356,A -85,B 0,C 180,E1 -11324.419,E2 -11324.419} C_VEL
LIN {X 0,Y 401.282,Z 925.871,A -85,B 0,C 180,E1 -11324.68,E2 -11324.68} C_VEL
LIN {X 0,Y 400.15,Z 977.715,A -85,B 0,C 180,E1 -11325.896,E2 -11325.896} C_VEL
LIN {X 0,Y 399.808,Z 988.93,A -85,B 0,C 180,E1 -11326.337,E2 -11326.337} C_VEL
LIN {X 0,Y 399.328,Z 998.777,A -85,B 0,C 180,E1 -11326.904,E2 -11326.904} C_VEL
LIN {X 0,Y 398.96,Z 1007.289,A -85,B 0,C 180,E1 -11327.538,E2 -11327.538} C_VEL
LIN {X 0,Y 398.557,Z 1015.531,A -85,B 0,C 180,E1 -11328.3,E2 -11328.3} C_VEL
LIN {X 0,Y 398.051,Z 1023.379,A -85,B 0,C 180,E1 -11329.188,E2 -11329.188} C_VEL
LIN {X 0,Y 397.603,Z 1029.868,A -85,B 0,C 180,E1 -11330.077,E2 -11330.077} C_VEL
LIN {X 0,Y 397.151,Z 1036.044,A -85,B 0,C 180,E1 -11331.093,E2 -11331.093} C_VEL
LIN {X 0,Y 396.774,Z 1042.347,A -85,B 0,C 180,E1 -11332.367,E2 -11332.367} C_VEL
LIN {X 0,Y 396.437,Z 1048.122,A -85,B 0,C 180,E1 -11333.894,E2 -11333.894} C_VEL
LIN {X 0,Y 396.102,Z 1051.146,A -85,B 0,C 180,E1 -11334.911,E2 -11334.911} C_VEL
LIN {X 0,Y 396.082,Z 1053.474,A -85,B 0,C 180,E1 -11335.93,E2 -11335.93} C_VEL
LIN {X 0,Y 396.036,Z 1055.189,A -85,B 0,C 180,E1 -11336.949,E2 -11336.949} C_VEL
LIN {X 0,Y 395.902,Z 1056.385,A -85,B 0,C 180,E1 -11337.966,E2 -11337.966} C_VEL
LIN {X 0,Y 395.814,Z 1057.075,A -85,B 0,C 180,E1 -11338.983,E2 -11338.983} C_VEL
LIN {X 0,Y 395.796,Z 1057.266,A -85,B 0,C 180,E1 -11340,E2 -11340} C_VEL
LIN {X 0,Y 395.813,Z 1056.88,A -85,B 0,C 180,E1 -11341.018,E2 -11341.018} C_VEL
LIN {X 0,Y 395.89,Z 1055.906,A -85,B 0,C 180,E1 -11342.035,E2 -11342.035} C_VEL
LIN {X 0,Y 395.921,Z 1053.547,A -85,B 0,C 180,E1 -11343.562,E2 -11343.562} C_VEL
LIN {X 0,Y 396.077,Z 1049.78,A -85,B 0,C 180,E1 -11345.09,E2 -11345.09} C_VEL
LIN {X 0,Y 396.331,Z 1045.096,A -85,B 0,C 180,E1 -11346.476,E2 -11346.476} C_VEL
LIN {X 0,Y 396.531,Z 1040.122,A -85,B 0,C 180,E1 -11347.639,E2 -11347.639} C_VEL
LIN {X 0,Y 396.794,Z 1034.805,A -85,B 0,C 180,E1 -11348.659,E2 -11348.659} C_VEL
LIN {X 0,Y 397.192,Z 1028.394,A -85,B 0,C 180,E1 -11349.678,E2 -11349.678} C_VEL
LIN {X 0,Y 397.653,Z 1020.608,A -85,B 0,C 180,E1 -11350.695,E2 -11350.695} C_VEL
LIN {X 0,Y 398.158,Z 1010.903,A -85,B 0,C 180,E1 -11351.712,E2 -11351.712} C_VEL
LIN {X 0,Y 398.595,Z 1001.422,A -85,B 0,C 180,E1 -11352.474,E2 -11352.474} C_VEL
LIN {X 0,Y 398.901,Z 992.328,A -85,B 0,C 180,E1 -11353.047,E2 -11353.047} C_VEL
LIN {X 0,Y 399.1,Z 982.932,A -85,B 0,C 180,E1 -11353.494,E2 -11353.494} C_VEL
LIN {X 0,Y 399.407,Z 973.295,A -85,B 0,C 180,E1 -11353.807,E2 -11353.807} C_VEL
LIN {X 0,Y 400.254,Z 915.739,A -85,B 0,C 180,E1 -11355.042,E2 -11355.042} C_VEL
LIN {X 0,Y 397.326,Z 898.628,A -85,B 0,C 180,E1 -11355.518,E2 -11355.518} C_VEL
LIN {X 0,Y 397.628,Z 890.274,A -85,B 0,C 180,E1 -11358.018,E2 -11358.018} C_VEL
LIN {X 0,Y 397.206,Z 885.818,A -85,B 0,C 180,E1 -11359.443,E2 -11359.443} C_VEL
LIN {X 0,Y 397.089,Z 885.837,A -85,B 0,C 180,E1 -11363.025,E2 -11363.025} C_VEL
LIN {X 0,Y 397.071,Z 885.833,A -85,B 0,C 180,E1 -11366.263,E2 -11366.263} C_VEL
LIN {X 0,Y 397.096,Z 885.831,A -85,B 0,C 180,E1 -11369.862,E2 -11369.862} C_VEL
LIN {X 0,Y 397.113,Z 885.831,A -85,B 0,C 180,E1 -11373.274,E2 -11373.274} C_VEL
LIN {X 0,Y 397.098,Z 885.835,A -85,B 0,C 180,E1 -11375.736,E2 -11375.736} C_VEL
LIN {X 0,Y 397.092,Z 885.83,A -85,B 0,C 180,E1 -11378.855,E2 -11378.855} C_VEL
LIN {X 0,Y 397.055,Z 885.838,A -85,B 0,C 180,E1 -11382.27,E2 -11382.27} C_VEL
LIN {X 0,Y 397.086,Z 885.831,A -85,B 0,C 180,E1 -11385.07,E2 -11385.07} C_VEL
LIN {X 0,Y 397.053,Z 885.84,A -85,B 0,C 180,E1 -11388.024,E2 -11388.024} C_VEL
LIN {X 0,Y 397.088,Z 885.832,A -85,B 0,C 180,E1 -11391.723,E2 -11391.723} C_VEL
LIN {X 0,Y 397.121,Z 885.826,A -85,B 0,C 180,E1 -11395.506,E2 -11395.506} C_VEL
LIN {X 0,Y 397.075,Z 885.834,A -85,B 0,C 180,E1 -11399.117,E2 -11399.117} C_VEL
LIN {X 0,Y 397.061,Z 885.835,A -85,B 0,C 180,E1 -11402.253,E2 -11402.253} C_VEL
LIN {X 0,Y 397.105,Z 885.835,A -85,B 0,C 180,E1 -11404.865,E2 -11404.865} C_VEL
LIN {X 0,Y 397.094,Z 885.83,A -85,B 0,C 180,E1 -11408.181,E2 -11408.181} C_VEL
LIN {X 0,Y 397.107,Z 885.833,A -85,B 0,C 180,E1 -11411.424,E2 -11411.424} C_VEL
LIN {X 0,Y 397.171,Z 885.821,A -85,B 0,C 180,E1 -11414.608,E2 -11414.608} C_VEL
LIN {X 0,Y 397.216,Z 885.819,A -85,B 0,C 180,E1 -11417.742,E2 -11417.742} C_VEL
LIN {X 0,Y 397.23,Z 885.813,A -85,B 0,C 180,E1 -11420.838,E2 -11420.838} C_VEL
LIN {X 0,Y 397.324,Z 885.807,A -85,B 0,C 180,E1 -11423.908,E2 -11423.908} C_VEL
LIN {X 0,Y 397.437,Z 885.794,A -85,B 0,C 180,E1 -11427.973,E2 -11427.973} C_VEL
LIN {X 0,Y 397.322,Z 885.801,A -85,B 0,C 180,E1 -11431.014,E2 -11431.014} C_VEL
LIN {X 0,Y 397.286,Z 885.806,A -85,B 0,C 180,E1 -11433.042,E2 -11433.042} C_VEL
LIN {X 0,Y 397.324,Z 885.805,A -85,B 0,C 180,E1 -11436.092,E2 -11436.092} C_VEL
LIN {X 0,Y 397.23,Z 885.813,A -85,B 0,C 180,E1 -11439.163,E2 -11439.163} C_VEL
LIN {X 0,Y 397.216,Z 885.818,A -85,B 0,C 180,E1 -11442.258,E2 -11442.258} C_VEL
LIN {X 0,Y 397.115,Z 885.828,A -85,B 0,C 180,E1 -11445.395,E2 -11445.395} C_VEL
LIN {X 0,Y 397.105,Z 885.828,A -85,B 0,C 180,E1 -11445.672,E2 -11445.672} C_VEL
LIN {X 0,Y 396.437,Z 885.917,A -85,B 0,C 180,E1 -11446.518,E2 -11446.518} C_VEL
LIN {X 0,Y 393.595,Z 886.266,A -85,B 0,C 180,E1 -11447.894,E2 -11447.894} C_VEL
LIN {X 0,Y 391.19,Z 886.571,A -85,B 0,C 180,E1 -11449.005,E2 -11449.005} C_VEL
LIN {X 0,Y 390.157,Z 886.694,A -85,B 0,C 180,E1 -11449.864,E2 -11449.864} C_VEL
LIN {X 0,Y 390.073,Z 886.705,A -85,B 0,C 180,E1 -11450.155,E2 -11450.155} C_VEL
LIN {X 0,Y 390.058,Z 886.71,A -85,B 0,C 180,E1 -11453.353,E2 -11453.353} C_VEL
LIN {X 0,Y 390.03,Z 886.712,A -85,B 0,C 180,E1 -11456.775,E2 -11456.775} C_VEL
LIN {X 0,Y 390.038,Z 886.709,A -85,B 0,C 180,E1 -11460.3,E2 -11460.3} C_VEL
LIN {X 0,Y 390.074,Z 886.706,A -85,B 0,C 180,E1 -11464.024,E2 -11464.024} C_VEL
LIN {X 0,Y 390.039,Z 886.715,A -85,B 0,C 180,E1 -11467.781,E2 -11467.781} C_VEL
LIN {X 0,Y 390.02,Z 886.711,A -85,B 0,C 180,E1 -11470.814,E2 -11470.814} C_VEL
LIN {X 0,Y 390.047,Z 886.713,A -85,B 0,C 180,E1 -11473.884,E2 -11473.884} C_VEL
LIN {X 0,Y 390.05,Z 886.708,A -85,B 0,C 180,E1 -11476.788,E2 -11476.788} C_VEL
LIN {X 0,Y 390.013,Z 886.713,A -85,B 0,C 180,E1 -11479.554,E2 -11479.554} C_VEL
LIN {X 0,Y 390.039,Z 886.715,A -85,B 0,C 180,E1 -11482.451,E2 -11482.451} C_VEL
LIN {X 0,Y 390.065,Z 886.707,A -85,B 0,C 180,E1 -11486.044,E2 -11486.044} C_VEL
LIN {X 0,Y 390.044,Z 886.708,A -85,B 0,C 180,E1 -11489.87,E2 -11489.87} C_VEL
LIN {X 0,Y 390.029,Z 886.712,A -85,B 0,C 180,E1 -11493.225,E2 -11493.225} C_VEL
LIN {X 0,Y 390.06,Z 886.71,A -85,B 0,C 180,E1 -11496.768,E2 -11496.768} C_VEL
LIN {X 0,Y 390.075,Z 886.704,A -85,B 0,C 180,E1 -11499.981,E2 -11499.981} C_VEL
LIN {X 0,Y 390.107,Z 886.706,A -85,B 0,C 180,E1 -11503.246,E2 -11503.246} C_VEL
LIN {X 0,Y 390.176,Z 886.692,A -85,B 0,C 180,E1 -11506.575,E2 -11506.575} C_VEL
LIN {X 0,Y 390.156,Z 886.701,A -85,B 0,C 180,E1 -11509.622,E2 -11509.622} C_VEL
LIN {X 0,Y 390.249,Z 886.682,A -85,B 0,C 180,E1 -11512.757,E2 -11512.757} C_VEL
LIN {X 0,Y 390.198,Z 886.689,A -85,B 0,C 180,E1 -11514.833,E2 -11514.833} C_VEL
LIN {X 0,Y 390.401,Z 886.67,A -85,B 0,C 180,E1 -11517.936,E2 -11517.936} C_VEL
LIN {X 0,Y 390.29,Z 886.677,A -85,B 0,C 180,E1 -11521.031,E2 -11521.031} C_VEL
LIN {X 0,Y 390.4,Z 886.67,A -85,B 0,C 180,E1 -11522.063,E2 -11522.063} C_VEL
LIN {X 0,Y 390.277,Z 886.685,A -85,B 0,C 180,E1 -11526.202,E2 -11526.202} C_VEL
LIN {X 0,Y 390.186,Z 886.69,A -85,B 0,C 180,E1 -11529.329,E2 -11529.329} C_VEL
LIN {X 0,Y 390.167,Z 886.698,A -85,B 0,C 180,E1 -11532.483,E2 -11532.483} C_VEL
LIN {X 0,Y 390.058,Z 886.706,A -85,B 0,C 180,E1 -11535.68,E2 -11535.68} C_VEL
LIN {X 0,Y 390.063,Z 886.705,A -85,B 0,C 180,E1 -11537.836,E2 -11537.836} C_VEL
LIN {X 0,Y 390.05,Z 886.712,A -85,B 0,C 180,E1 -11541.122,E2 -11541.122} C_VEL
LIN {X 0,Y 390.036,Z 886.71,A -85,B 0,C 180,E1 -11544.483,E2 -11544.483} C_VEL
LIN {X 0,Y 390.016,Z 886.712,A -85,B 0,C 180,E1 -11547.997,E2 -11547.997} C_VEL
LIN {X 0,Y 390.017,Z 886.718,A -85,B 0,C 180,E1 -11551.505,E2 -11551.505} C_VEL
LIN {X 0,Y 390.067,Z 886.708,A -85,B 0,C 180,E1 -11555.208,E2 -11555.208} C_VEL
LIN {X 0,Y 390.055,Z 886.707,A -85,B 0,C 180,E1 -11559.096,E2 -11559.096} C_VEL
LIN {X 0,Y 390.028,Z 886.712,A -85,B 0,C 180,E1 -11562.371,E2 -11562.371} C_VEL
LIN {X 0,Y 390.039,Z 886.709,A -85,B 0,C 180,E1 -11565.353,E2 -11565.353} C_VEL
LIN {X 0,Y 390.013,Z 886.719,A -85,B 0,C 180,E1 -11568.184,E2 -11568.184} C_VEL
LIN {X 0,Y 390.053,Z 886.708,A -85,B 0,C 180,E1 -11570.903,E2 -11570.903} C_VEL
LIN {X 0,Y 390.07,Z 886.708,A -85,B 0,C 180,E1 -11574.791,E2 -11574.791} C_VEL
LIN {X 0,Y 390.017,Z 886.716,A -85,B 0,C 180,E1 -11578.495,E2 -11578.495} C_VEL
LIN {X 0,Y 390.014,Z 886.712,A -85,B 0,C 180,E1 -11582.003,E2 -11582.003} C_VEL
LIN {X 0,Y 390.095,Z 886.775,A -85,B 0,C 180,E1 -11583.762,E2 -11583.762} C_VEL
LIN {X 0,Y 392.209,Z 898.321,A -85,B 0,C 180,E1 -11586.782,E2 -11586.782} C_VEL
LIN {X 0,Y 391.673,Z 908.351,A -85,B 0,C 180,E1 -11589.244,E2 -11589.244} C_VEL
LIN {X 0,Y 390.604,Z 923.223,A -85,B 0,C 180,E1 -11592.836,E2 -11592.836} C_VEL
LIN {X 0,Y 390.315,Z 929.032,A -85,B 0,C 180,E1 -11594.23,E2 -11594.23} C_VEL
LIN {X 0,Y 393.13,Z 954.275,A -85,B 0,C 180,E1 -11594.9,E2 -11594.9} C_VEL
LIN {X 0,Y 392.357,Z 1007.887,A -85,B 0,C 180,E1 -11596.105,E2 -11596.105} C_VEL
LIN {X 0,Y 391.867,Z 1020.086,A -85,B 0,C 180,E1 -11596.583,E2 -11596.583} C_VEL
LIN {X 0,Y 391.456,Z 1029.978,A -85,B 0,C 180,E1 -11597.163,E2 -11597.163} C_VEL
LIN {X 0,Y 391.038,Z 1038.527,A -85,B 0,C 180,E1 -11597.808,E2 -11597.808} C_VEL
LIN {X 0,Y 390.554,Z 1046.779,A -85,B 0,C 180,E1 -11598.583,E2 -11598.583} C_VEL
LIN {X 0,Y 390.12,Z 1054.651,A -85,B 0,C 180,E1 -11599.49,E2 -11599.49} C_VEL
LIN {X 0,Y 389.666,Z 1062.91,A -85,B 0,C 180,E1 -11600.658,E2 -11600.658} C_VEL
LIN {X 0,Y 389.28,Z 1070.11,A -85,B 0,C 180,E1 -11601.957,E2 -11601.957} C_VEL
LIN {X 0,Y 389.046,Z 1075.802,A -85,B 0,C 180,E1 -11603.257,E2 -11603.257} C_VEL
LIN {X 0,Y 388.857,Z 1081.076,A -85,B 0,C 180,E1 -11604.815,E2 -11604.815} C_VEL
LIN {X 0,Y 388.712,Z 1084.894,A -85,B 0,C 180,E1 -11606.372,E2 -11606.372} C_VEL
LIN {X 0,Y 388.746,Z 1087.276,A -85,B 0,C 180,E1 -11607.928,E2 -11607.928} C_VEL
LIN {X 0,Y 388.739,Z 1088.224,A -85,B 0,C 180,E1 -11608.964,E2 -11608.964} C_VEL
LIN {X 0,Y 388.723,Z 1088.548,A -85,B 0,C 180,E1 -11610,E2 -11610} C_VEL
LIN {X 0,Y 388.737,Z 1088.337,A -85,B 0,C 180,E1 -11611.036,E2 -11611.036} C_VEL
LIN {X 0,Y 388.713,Z 1087.618,A -85,B 0,C 180,E1 -11612.072,E2 -11612.072} C_VEL
LIN {X 0,Y 388.687,Z 1086.386,A -85,B 0,C 180,E1 -11613.109,E2 -11613.109} C_VEL
LIN {X 0,Y 388.833,Z 1083.396,A -85,B 0,C 180,E1 -11614.665,E2 -11614.665} C_VEL
LIN {X 0,Y 388.92,Z 1079.077,A -85,B 0,C 180,E1 -11616.224,E2 -11616.224} C_VEL
LIN {X 0,Y 389.254,Z 1073.234,A -85,B 0,C 180,E1 -11617.782,E2 -11617.782} C_VEL
LIN {X 0,Y 389.61,Z 1066.837,A -85,B 0,C 180,E1 -11619.081,E2 -11619.081} C_VEL
LIN {X 0,Y 390.051,Z 1060.597,A -85,B 0,C 180,E1 -11620.118,E2 -11620.118} C_VEL
LIN {X 0,Y 390.607,Z 1053.021,A -85,B 0,C 180,E1 -11621.152,E2 -11621.152} C_VEL
LIN {X 0,Y 391.125,Z 1044.988,A -85,B 0,C 180,E1 -11622.057,E2 -11622.057} C_VEL
LIN {X 0,Y 391.718,Z 1035.076,A -85,B 0,C 180,E1 -11622.96,E2 -11622.96} C_VEL
LIN {X 0,Y 392.332,Z 1023.666,A -85,B 0,C 180,E1 -11623.73,E2 -11623.73} C_VEL
LIN {X 0,Y 392.897,Z 1013.975,A -85,B 0,C 180,E1 -11624.205,E2 -11624.205} C_VEL
LIN {X 0,Y 393.324,Z 1003.764,A -85,B 0,C 180,E1 -11624.554,E2 -11624.554} C_VEL
LIN {X 0,Y 394.2,Z 952.466,A -85,B 0,C 180,E1 -11625.779,E2 -11625.779} C_VEL
LIN {X 0,Y 392.431,Z 936.859,A -85,B 0,C 180,E1 -11626.286,E2 -11626.286} C_VEL
LIN {X 0,Y 390.707,Z 927.002,A -85,B 0,C 180,E1 -11626.671,E2 -11626.671} C_VEL
LIN {X 0,Y 391.85,Z 911.899,A -85,B 0,C 180,E1 -11630.471,E2 -11630.471} C_VEL
LIN {X 0,Y 392.758,Z 902.576,A -85,B 0,C 180,E1 -11632.904,E2 -11632.904} C_VEL
LIN {X 0,Y 392.262,Z 897.557,A -85,B 0,C 180,E1 -11634.336,E2 -11634.336} C_VEL
LIN {X 0,Y 390.725,Z 889.854,A -85,B 0,C 180,E1 -11636.723,E2 -11636.723} C_VEL
LIN {X 0,Y 390.013,Z 886.72,A -85,B 0,C 180,E1 -11637.792,E2 -11637.792} C_VEL
LIN {X 0,Y 390.032,Z 886.714,A -85,B 0,C 180,E1 -11640.3,E2 -11640.3} C_VEL
LIN {X 0,Y 390.067,Z 886.711,A -85,B 0,C 180,E1 -11644.025,E2 -11644.025} C_VEL
LIN {X 0,Y 390.031,Z 886.715,A -85,B 0,C 180,E1 -11647.781,E2 -11647.781} C_VEL
LIN {X 0,Y 390.013,Z 886.713,A -85,B 0,C 180,E1 -11650.814,E2 -11650.814} C_VEL
LIN {X 0,Y 390.041,Z 886.713,A -85,B 0,C 180,E1 -11653.884,E2 -11653.884} C_VEL
LIN {X 0,Y 390.043,Z 886.71,A -85,B 0,C 180,E1 -11656.788,E2 -11656.788} C_VEL
LIN {X 0,Y 390.007,Z 886.716,A -85,B 0,C 180,E1 -11659.555,E2 -11659.555} C_VEL
LIN {X 0,Y 390.033,Z 886.715,A -85,B 0,C 180,E1 -11662.451,E2 -11662.451} C_VEL
LIN {X 0,Y 390.06,Z 886.712,A -85,B 0,C 180,E1 -11666.045,E2 -11666.045} C_VEL
LIN {X 0,Y 390.039,Z 886.713,A -85,B 0,C 180,E1 -11669.871,E2 -11669.871} C_VEL
LIN {X 0,Y 390.024,Z 886.717,A -85,B 0,C 180,E1 -11673.226,E2 -11673.226} C_VEL
LIN {X 0,Y 390.054,Z 886.718,A -85,B 0,C 180,E1 -11676.768,E2 -11676.768} C_VEL
LIN {X 0,Y 390.069,Z 886.897,A -85,B 0,C 180,E1 -11678.186,E2 -11678.186} C_VEL
LIN {X 0,Y 391.265,Z 893.067,A -85,B 0,C 180,E1 -11680.592,E2 -11680.592} C_VEL
LIN {X 0,Y 391.504,Z 897.648,A -85,B 0,C 180,E1 -11682.232,E2 -11682.232} C_VEL
LIN {X 0,Y 391.206,Z 901.278,A -85,B 0,C 180,E1 -11683.457,E2 -11683.457} C_VEL
LIN {X 0,Y 394.567,Z 915.605,A -85,B 0,C 180,E1 -11684.046,E2 -11684.046} C_VEL
LIN {X 0,Y 394.782,Z 919.557,A -85,B 0,C 180,E1 -11684.163,E2 -11684.163} C_VEL
LIN {X 0,Y 393.411,Z 978.01,A -85,B 0,C 180,E1 -11685.583,E2 -11685.583} C_VEL
LIN {X 0,Y 393.052,Z 989.226,A -85,B 0,C 180,E1 -11686.032,E2 -11686.032} C_VEL
LIN {X 0,Y 392.508,Z 999.985,A -85,B 0,C 180,E1 -11686.672,E2 -11686.672} C_VEL
LIN {X 0,Y 392.1,Z 1008.315,A -85,B 0,C 180,E1 -11687.317,E2 -11687.317} C_VEL
LIN {X 0,Y 391.655,Z 1016.397,A -85,B 0,C 180,E1 -11688.091,E2 -11688.091} C_VEL
LIN {X 0,Y 391.121,Z 1024.126,A -85,B 0,C 180,E1 -11688.994,E2 -11688.994} C_VEL
LIN {X 0,Y 390.539,Z 1032.232,A -85,B 0,C 180,E1 -11690.157,E2 -11690.157} C_VEL
LIN {X 0,Y 389.97,Z 1039.327,A -85,B 0,C 180,E1 -11691.45,E2 -11691.45} C_VEL
LIN {X 0,Y 389.615,Z 1045.126,A -85,B 0,C 180,E1 -11692.797,E2 -11692.797} C_VEL
LIN {X 0,Y 389.211,Z 1050.145,A -85,B 0,C 180,E1 -11694.301,E2 -11694.301} C_VEL
LIN {X 0,Y 389.009,Z 1053.914,A -85,B 0,C 180,E1 -11695.856,E2 -11695.856} C_VEL
LIN {X 0,Y 388.98,Z 1055.597,A -85,B 0,C 180,E1 -11696.893,E2 -11696.893} C_VEL
LIN {X 0,Y 388.84,Z 1056.752,A -85,B 0,C 180,E1 -11697.929,E2 -11697.929} C_VEL
LIN {X 0,Y 388.745,Z 1057.399,A -85,B 0,C 180,E1 -11698.965,E2 -11698.965} C_VEL
LIN {X 0,Y 388.724,Z 1057.543,A -85,B 0,C 180,E1 -11700,E2 -11700} C_VEL
LIN {X 0,Y 388.744,Z 1057.141,A -85,B 0,C 180,E1 -11701.036,E2 -11701.036} C_VEL
LIN {X 0,Y 388.806,Z 1056.133,A -85,B 0,C 180,E1 -11702.072,E2 -11702.072} C_VEL
LIN {X 0,Y 388.832,Z 1053.703,A -85,B 0,C 180,E1 -11703.628,E2 -11703.628} C_VEL
LIN {X 0,Y 389.002,Z 1049.848,A -85,B 0,C 180,E1 -11705.183,E2 -11705.183} C_VEL
LIN {X 0,Y 389.292,Z 1044.72,A -85,B 0,C 180,E1 -11706.693,E2 -11706.693} C_VEL
LIN {X 0,Y 389.476,Z 1040.055,A -85,B 0,C 180,E1 -11707.779,E2 -11707.779} C_VEL
LIN {X 0,Y 389.77,Z 1034.661,A -85,B 0,C 180,E1 -11708.817,E2 -11708.817} C_VEL
LIN {X 0,Y 390.191,Z 1028.165,A -85,B 0,C 180,E1 -11709.853,E2 -11709.853} C_VEL
LIN {X 0,Y 390.708,Z 1019.217,A -85,B 0,C 180,E1 -11711.019,E2 -11711.019} C_VEL
LIN {X 0,Y 391.166,Z 1010.316,A -85,B 0,C 180,E1 -11711.925,E2 -11711.925} C_VEL
LIN {X 0,Y 391.595,Z 1000.625,A -85,B 0,C 180,E1 -11712.701,E2 -11712.701} C_VEL
LIN {X 0,Y 391.98,Z 991.262,A -85,B 0,C 180,E1 -11713.281,E2 -11713.281} C_VEL
LIN {X 0,Y 392.194,Z 981.441,A -85,B 0,C 180,E1 -11713.736,E2 -11713.736} C_VEL
LIN {X 0,Y 392.551,Z 968.089,A -85,B 0,C 180,E1 -11714.119,E2 -11714.119} C_VEL
LIN {X 0,Y 393.24,Z 916.203,A -85,B 0,C 180,E1 -11715.254,E2 -11715.254} C_VEL
LIN {X 0,Y 390.316,Z 898.777,A -85,B 0,C 180,E1 -11715.771,E2 -11715.771} C_VEL
LIN {X 0,Y 390.605,Z 892.053,A -85,B 0,C 180,E1 -11717.811,E2 -11717.811} C_VEL
LIN {X 0,Y 390.162,Z 886.695,A -85,B 0,C 180,E1 -11719.535,E2 -11719.535} C_VEL
LIN {X 0,Y 390.054,Z 886.71,A -85,B 0,C 180,E1 -11723.354,E2 -11723.354} C_VEL
LIN {X 0,Y 390.027,Z 886.712,A -85,B 0,C 180,E1 -11726.775,E2 -11726.775} C_VEL
LIN {X 0,Y 390.035,Z 886.709,A -85,B 0,C 180,E1 -11730.301,E2 -11730.301} C_VEL
LIN {X 0,Y 390.071,Z 886.707,A -85,B 0,C 180,E1 -11734.025,E2 -11734.025} C_VEL
LIN {X 0,Y 390.039,Z 886.714,A -85,B 0,C 180,E1 -11737.55,E2 -11737.55} C_VEL
LIN {X 0,Y 390.018,Z 886.711,A -85,B 0,C 180,E1 -11740.815,E2 -11740.815} C_VEL
LIN {X 0,Y 390.045,Z 886.713,A -85,B 0,C 180,E1 -11743.885,E2 -11743.885} C_VEL
LIN {X 0,Y 390.049,Z 886.708,A -85,B 0,C 180,E1 -11746.789,E2 -11746.789} C_VEL
LIN {X 0,Y 390.012,Z 886.713,A -85,B 0,C 180,E1 -11749.555,E2 -11749.555} C_VEL
LIN {X 0,Y 390.039,Z 886.715,A -85,B 0,C 180,E1 -11752.451,E2 -11752.451} C_VEL
LIN {X 0,Y 390.065,Z 886.707,A -85,B 0,C 180,E1 -11756.045,E2 -11756.045} C_VEL
LIN {X 0,Y 390.044,Z 886.708,A -85,B 0,C 180,E1 -11759.871,E2 -11759.871} C_VEL
LIN {X 0,Y 390.029,Z 886.713,A -85,B 0,C 180,E1 -11763.226,E2 -11763.226} C_VEL
LIN {X 0,Y 390.062,Z 886.71,A -85,B 0,C 180,E1 -11766.767,E2 -11766.767} C_VEL
LIN {X 0,Y 390.075,Z 886.704,A -85,B 0,C 180,E1 -11769.982,E2 -11769.982} C_VEL
LIN {X 0,Y 390.129,Z 886.704,A -85,B 0,C 180,E1 -11773.248,E2 -11773.248} C_VEL
LIN {X 0,Y 390.2,Z 886.689,A -85,B 0,C 180,E1 -11776.562,E2 -11776.562} C_VEL
LIN {X 0,Y 390.188,Z 886.69,A -85,B 0,C 180,E1 -11780.671,E2 -11780.671} C_VEL
LIN {X 0,Y 390.279,Z 886.686,A -85,B 0,C 180,E1 -11783.798,E2 -11783.798} C_VEL
LIN {X 0,Y 390.403,Z 886.67,A -85,B 0,C 180,E1 -11787.937,E2 -11787.937} C_VEL
LIN {X 0,Y 390.293,Z 886.677,A -85,B 0,C 180,E1 -11791.032,E2 -11791.032} C_VEL
LIN {X 0,Y 390.402,Z 886.669,A -85,B 0,C 180,E1 -11792.064,E2 -11792.064} C_VEL
LIN {X 0,Y 390.28,Z 886.684,A -85,B 0,C 180,E1 -11796.203,E2 -11796.203} C_VEL
LIN {X 0,Y 390.188,Z 886.69,A -85,B 0,C 180,E1 -11799.329,E2 -11799.329} C_VEL
LIN {X 0,Y 390.17,Z 886.698,A -85,B 0,C 180,E1 -11802.483,E2 -11802.483} C_VEL
LIN {X 0,Y 390.06,Z 886.706,A -85,B 0,C 180,E1 -11805.68,E2 -11805.68} C_VEL
LIN {X 0,Y 390.067,Z 886.705,A -85,B 0,C 180,E1 -11807.836,E2 -11807.836} C_VEL
LIN {X 0,Y 390.073,Z 886.705,A -85,B 0,C 180,E1 -11810.155,E2 -11810.155} C_VEL
LIN {X 0,Y 389.396,Z 886.795,A -85,B 0,C 180,E1 -11811.017,E2 -11811.017} C_VEL
LIN {X 0,Y 386.513,Z 887.149,A -85,B 0,C 180,E1 -11812.417,E2 -11812.417} C_VEL
LIN {X 0,Y 384.084,Z 887.452,A -85,B 0,C 180,E1 -11813.549,E2 -11813.549} C_VEL
LIN {X 0,Y 383.055,Z 887.579,A -85,B 0,C 180,E1 -11814.424,E2 -11814.424} C_VEL
LIN {X 0,Y 382.979,Z 887.59,A -85,B 0,C 180,E1 -11814.721,E2 -11814.721} C_VEL
LIN {X 0,Y 382.983,Z 887.587,A -85,B 0,C 180,E1 -11818.255,E2 -11818.255} C_VEL
LIN {X 0,Y 382.982,Z 887.59,A -85,B 0,C 180,E1 -11820.919,E2 -11820.919} C_VEL
LIN {X 0,Y 383.015,Z 887.584,A -85,B 0,C 180,E1 -11824.669,E2 -11824.669} C_VEL
LIN {X 0,Y 382.995,Z 887.591,A -85,B 0,C 180,E1 -11827.902,E2 -11827.902} C_VEL
LIN {X 0,Y 382.964,Z 887.592,A -85,B 0,C 180,E1 -11831.35,E2 -11831.35} C_VEL
LIN {X 0,Y 382.992,Z 887.59,A -85,B 0,C 180,E1 -11834.302,E2 -11834.302} C_VEL
LIN {X 0,Y 382.986,Z 887.587,A -85,B 0,C 180,E1 -11837.236,E2 -11837.236} C_VEL
LIN {X 0,Y 382.987,Z 887.592,A -85,B 0,C 180,E1 -11840.419,E2 -11840.419} C_VEL
LIN {X 0,Y 383.018,Z 887.586,A -85,B 0,C 180,E1 -11844.043,E2 -11844.043} C_VEL
LIN {X 0,Y 382.987,Z 887.587,A -85,B 0,C 180,E1 -11847.579,E2 -11847.579} C_VEL
LIN {X 0,Y 382.977,Z 887.591,A -85,B 0,C 180,E1 -11850.298,E2 -11850.298} C_VEL
LIN {X 0,Y 383.006,Z 887.585,A -85,B 0,C 180,E1 -11854.045,E2 -11854.045} C_VEL
LIN {X 0,Y 382.987,Z 887.59,A -85,B 0,C 180,E1 -11857.333,E2 -11857.333} C_VEL
LIN {X 0,Y 383.021,Z 887.585,A -85,B 0,C 180,E1 -11860.714,E2 -11860.714} C_VEL
LIN {X 0,Y 383.015,Z 887.584,A -85,B 0,C 180,E1 -11864.023,E2 -11864.023} C_VEL
LIN {X 0,Y 383.13,Z 887.574,A -85,B 0,C 180,E1 -11867.283,E2 -11867.283} C_VEL
LIN {X 0,Y 383.137,Z 887.568,A -85,B 0,C 180,E1 -11870.497,E2 -11870.497} C_VEL
LIN {X 0,Y 383.236,Z 887.562,A -85,B 0,C 180,E1 -11873.682,E2 -11873.682} C_VEL
LIN {X 0,Y 383.366,Z 887.546,A -85,B 0,C 180,E1 -11877.898,E2 -11877.898} C_VEL
LIN {X 0,Y 383.262,Z 887.553,A -85,B 0,C 180,E1 -11881.05,E2 -11881.05} C_VEL
LIN {X 0,Y 383.365,Z 887.547,A -85,B 0,C 180,E1 -11882.101,E2 -11882.101} C_VEL
LIN {X 0,Y 383.235,Z 887.563,A -85,B 0,C 180,E1 -11886.317,E2 -11886.317} C_VEL
LIN {X 0,Y 383.136,Z 887.568,A -85,B 0,C 180,E1 -11889.502,E2 -11889.502} C_VEL
LIN {X 0,Y 383.13,Z 887.569,A -85,B 0,C 180,E1 -11893.537,E2 -11893.537} C_VEL
LIN {X 0,Y 383.054,Z 887.579,A -85,B 0,C 180,E1 -11897.434,E2 -11897.434} C_VEL
LIN {X 0,Y 383.015,Z 887.587,A -85,B 0,C 180,E1 -11900.64,E2 -11900.64} C_VEL
LIN {X 0,Y 383.005,Z 887.585,A -85,B 0,C 180,E1 -11903.809,E2 -11903.809} C_VEL
LIN {X 0,Y 382.966,Z 887.596,A -85,B 0,C 180,E1 -11907.308,E2 -11907.308} C_VEL
LIN {X 0,Y 382.978,Z 887.59,A -85,B 0,C 180,E1 -11910.919,E2 -11910.919} C_VEL
LIN {X 0,Y 383.01,Z 887.584,A -85,B 0,C 180,E1 -11914.668,E2 -11914.668} C_VEL
LIN {X 0,Y 382.991,Z 887.591,A -85,B 0,C 180,E1 -11917.901,E2 -11917.901} C_VEL
LIN {X 0,Y 382.959,Z 887.592,A -85,B 0,C 180,E1 -11921.35,E2 -11921.35} C_VEL
LIN {X 0,Y 382.988,Z 887.59,A -85,B 0,C 180,E1 -11924.302,E2 -11924.302} C_VEL
LIN {X 0,Y 382.981,Z 887.588,A -85,B 0,C 180,E1 -11927.236,E2 -11927.236} C_VEL
LIN {X 0,Y 382.982,Z 887.593,A -85,B 0,C 180,E1 -11930.419,E2 -11930.419} C_VEL
LIN {X 0,Y 383.014,Z 887.586,A -85,B 0,C 180,E1 -11934.043,E2 -11934.043} C_VEL
LIN {X 0,Y 382.982,Z 887.587,A -85,B 0,C 180,E1 -11937.579,E2 -11937.579} C_VEL
LIN {X 0,Y 382.972,Z 887.591,A -85,B 0,C 180,E1 -11940.298,E2 -11940.298} C_VEL
LIN {X 0,Y 383.047,Z 887.693,A -85,B 0,C 180,E1 -11943.618,E2 -11943.618} C_VEL
LIN {X 0,Y 385.132,Z 898.949,A -85,B 0,C 180,E1 -11946.615,E2 -11946.615} C_VEL
LIN {X 0,Y 384.889,Z 905.65,A -85,B 0,C 180,E1 -11948.299,E2 -11948.299} C_VEL
LIN {X 0,Y 383.865,Z 920.081,A -85,B 0,C 180,E1 -11951.865,E2 -11951.865} C_VEL
LIN {X 0,Y 383.312,Z 928.922,A -85,B 0,C 180,E1 -11954.002,E2 -11954.002} C_VEL
LIN {X 0,Y 386.179,Z 954.988,A -85,B 0,C 180,E1 -11954.707,E2 -11954.707} C_VEL
LIN {X 0,Y 385.388,Z 1007.076,A -85,B 0,C 180,E1 -11955.916,E2 -11955.916} C_VEL
LIN {X 0,Y 384.883,Z 1018.137,A -85,B 0,C 180,E1 -11956.335,E2 -11956.335} C_VEL
LIN {X 0,Y 384.526,Z 1028.509,A -85,B 0,C 180,E1 -11956.928,E2 -11956.928} C_VEL
LIN {X 0,Y 383.985,Z 1038.77,A -85,B 0,C 180,E1 -11957.715,E2 -11957.715} C_VEL
LIN {X 0,Y 383.494,Z 1046.927,A -85,B 0,C 180,E1 -11958.504,E2 -11958.504} C_VEL
LIN {X 0,Y 383.044,Z 1054.727,A -85,B 0,C 180,E1 -11959.427,E2 -11959.427} C_VEL
LIN {X 0,Y 382.532,Z 1063.713,A -85,B 0,C 180,E1 -11960.749,E2 -11960.749} C_VEL
LIN {X 0,Y 382.156,Z 1070.649,A -85,B 0,C 180,E1 -11962.072,E2 -11962.072} C_VEL
LIN {X 0,Y 381.999,Z 1075.208,A -85,B 0,C 180,E1 -11963.132,E2 -11963.132} C_VEL
LIN {X 0,Y 381.777,Z 1078.644,A -85,B 0,C 180,E1 -11964.078,E2 -11964.078} C_VEL
LIN {X 0,Y 381.771,Z 1082.055,A -85,B 0,C 180,E1 -11965.248,E2 -11965.248} C_VEL
LIN {X 0,Y 381.606,Z 1085.353,A -85,B 0,C 180,E1 -11966.833,E2 -11966.833} C_VEL
LIN {X 0,Y 381.647,Z 1086.908,A -85,B 0,C 180,E1 -11967.889,E2 -11967.889} C_VEL
LIN {X 0,Y 381.671,Z 1087.874,A -85,B 0,C 180,E1 -11968.945,E2 -11968.945} C_VEL
LIN {X 0,Y 381.653,Z 1088.226,A -85,B 0,C 180,E1 -11970,E2 -11970} C_VEL
LIN {X 0,Y 381.669,Z 1088.061,A -85,B 0,C 180,E1 -11971.055,E2 -11971.055} C_VEL
LIN {X 0,Y 381.612,Z 1087.381,A -85,B 0,C 180,E1 -11972.111,E2 -11972.111} C_VEL
LIN {X 0,Y 381.596,Z 1086.184,A -85,B 0,C 180,E1 -11973.167,E2 -11973.167} C_VEL
LIN {X 0,Y 381.745,Z 1083.224,A -85,B 0,C 180,E1 -11974.752,E2 -11974.752} C_VEL
LIN {X 0,Y 381.846,Z 1078.926,A -85,B 0,C 180,E1 -11976.34,E2 -11976.34} C_VEL
LIN {X 0,Y 382.144,Z 1074.184,A -85,B 0,C 180,E1 -11977.662,E2 -11977.662} C_VEL
LIN {X 0,Y 382.605,Z 1066.828,A -85,B 0,C 180,E1 -11979.249,E2 -11979.249} C_VEL
LIN {X 0,Y 383.061,Z 1060.673,A -85,B 0,C 180,E1 -11980.305,E2 -11980.305} C_VEL
LIN {X 0,Y 383.72,Z 1052.167,A -85,B 0,C 180,E1 -11981.489,E2 -11981.489} C_VEL
LIN {X 0,Y 384.304,Z 1044.024,A -85,B 0,C 180,E1 -11982.408,E2 -11982.408} C_VEL
LIN {X 0,Y 384.908,Z 1033.928,A -85,B 0,C 180,E1 -11983.327,E2 -11983.327} C_VEL
LIN {X 0,Y 385.545,Z 1023.303,A -85,B 0,C 180,E1 -11984.044,E2 -11984.044} C_VEL
LIN {X 0,Y 386.15,Z 1013.63,A -85,B 0,C 180,E1 -11984.526,E2 -11984.526} C_VEL
LIN {X 0,Y 386.565,Z 1003.918,A -85,B 0,C 180,E1 -11984.868,E2 -11984.868} C_VEL
LIN {X 0,Y 387.565,Z 953.2,A -85,B 0,C 180,E1 -11986.135,E2 -11986.135} C_VEL
LIN {X 0,Y 385.897,Z 938.328,A -85,B 0,C 180,E1 -11986.636,E2 -11986.636} C_VEL
LIN {X 0,Y 383.78,Z 926.724,A -85,B 0,C 180,E1 -11987.091,E2 -11987.091} C_VEL
LIN {X 0,Y 385.135,Z 911.143,A -85,B 0,C 180,E1 -11991.125,E2 -11991.125} C_VEL
LIN {X 0,Y 385.868,Z 903.967,A -85,B 0,C 180,E1 -11993.053,E2 -11993.053} C_VEL
LIN {X 0,Y 385.209,Z 898.056,A -85,B 0,C 180,E1 -11994.811,E2 -11994.811} C_VEL
LIN {X 0,Y 383.618,Z 890.513,A -85,B 0,C 180,E1 -11997.258,E2 -11997.258} C_VEL
LIN {X 0,Y 382.98,Z 887.595,A -85,B 0,C 180,E1 -11998.323,E2 -11998.323} C_VEL
LIN {X 0,Y 382.976,Z 887.595,A -85,B 0,C 180,E1 -12000.919,E2 -12000.919} C_VEL
LIN {X 0,Y 383.008,Z 887.59,A -85,B 0,C 180,E1 -12004.669,E2 -12004.669} C_VEL
LIN {X 0,Y 382.987,Z 887.592,A -85,B 0,C 180,E1 -12007.902,E2 -12007.902} C_VEL
LIN {X 0,Y 382.957,Z 887.595,A -85,B 0,C 180,E1 -12011.351,E2 -12011.351} C_VEL
LIN {X 0,Y 382.986,Z 887.593,A -85,B 0,C 180,E1 -12014.302,E2 -12014.302} C_VEL
LIN {X 0,Y 382.979,Z 887.59,A -85,B 0,C 180,E1 -12017.236,E2 -12017.236} C_VEL
LIN {X 0,Y 382.981,Z 887.591,A -85,B 0,C 180,E1 -12020.42,E2 -12020.42} C_VEL
LIN {X 0,Y 383.01,Z 887.588,A -85,B 0,C 180,E1 -12024.043,E2 -12024.043} C_VEL
LIN {X 0,Y 382.981,Z 887.592,A -85,B 0,C 180,E1 -12027.579,E2 -12027.579} C_VEL
LIN {X 0,Y 382.971,Z 887.595,A -85,B 0,C 180,E1 -12030.299,E2 -12030.299} C_VEL
LIN {X 0,Y 383.001,Z 887.591,A -85,B 0,C 180,E1 -12034.045,E2 -12034.045} C_VEL
LIN {X 0,Y 383.009,Z 887.66,A -85,B 0,C 180,E1 -12037.656,E2 -12037.656} C_VEL
LIN {X 0,Y 384.268,Z 894.001,A -85,B 0,C 180,E1 -12040.224,E2 -12040.224} C_VEL
LIN {X 0,Y 384.639,Z 898.494,A -85,B 0,C 180,E1 -12041.904,E2 -12041.904} C_VEL
LIN {X 0,Y 384.394,Z 901.696,A -85,B 0,C 180,E1 -12043.015,E2 -12043.015} C_VEL
LIN {X 0,Y 387.928,Z 916.425,A -85,B 0,C 180,E1 -12043.665,E2 -12043.665} C_VEL
LIN {X 0,Y 388.183,Z 920.854,A -85,B 0,C 180,E1 -12043.799,E2 -12043.799} C_VEL
LIN {X 0,Y 386.678,Z 978.592,A -85,B 0,C 180,E1 -12045.259,E2 -12045.259} C_VEL
LIN {X 0,Y 386.256,Z 990.752,A -85,B 0,C 180,E1 -12045.781,E2 -12045.781} C_VEL
LIN {X 0,Y 385.673,Z 1001.194,A -85,B 0,C 180,E1 -12046.431,E2 -12046.431} C_VEL
LIN {X 0,Y 385.187,Z 1010.835,A -85,B 0,C 180,E1 -12047.219,E2 -12047.219} C_VEL
LIN {X 0,Y 384.486,Z 1020.888,A -85,B 0,C 180,E1 -12048.267,E2 -12048.267} C_VEL
LIN {X 0,Y 383.858,Z 1029.582,A -85,B 0,C 180,E1 -12049.451,E2 -12049.451} C_VEL
LIN {X 0,Y 383.322,Z 1035.904,A -85,B 0,C 180,E1 -12050.503,E2 -12050.503} C_VEL
LIN {X 0,Y 382.892,Z 1041.149,A -85,B 0,C 180,E1 -12051.557,E2 -12051.557} C_VEL
LIN {X 0,Y 382.572,Z 1045.998,A -85,B 0,C 180,E1 -12052.748,E2 -12052.748} C_VEL
LIN {X 0,Y 382.181,Z 1050.644,A -85,B 0,C 180,E1 -12054.196,E2 -12054.196} C_VEL
LIN {X 0,Y 381.937,Z 1054.347,A -85,B 0,C 180,E1 -12055.779,E2 -12055.779} C_VEL
LIN {X 0,Y 381.906,Z 1056.007,A -85,B 0,C 180,E1 -12056.836,E2 -12056.836} C_VEL
LIN {X 0,Y 381.781,Z 1057.12,A -85,B 0,C 180,E1 -12057.891,E2 -12057.891} C_VEL
LIN {X 0,Y 381.678,Z 1057.723,A -85,B 0,C 180,E1 -12058.945,E2 -12058.945} C_VEL
LIN {X 0,Y 381.655,Z 1057.82,A -85,B 0,C 180,E1 -12060,E2 -12060} C_VEL
LIN {X 0,Y 381.677,Z 1057.39,A -85,B 0,C 180,E1 -12061.056,E2 -12061.056} C_VEL
LIN {X 0,Y 381.71,Z 1056.35,A -85,B 0,C 180,E1 -12062.111,E2 -12062.111} C_VEL
LIN {X 0,Y 381.747,Z 1053.826,A -85,B 0,C 180,E1 -12063.695,E2 -12063.695} C_VEL
LIN {X 0,Y 381.931,Z 1049.879,A -85,B 0,C 180,E1 -12065.28,E2 -12065.28} C_VEL
LIN {X 0,Y 382.235,Z 1044.569,A -85,B 0,C 180,E1 -12066.843,E2 -12066.843} C_VEL
LIN {X 0,Y 382.484,Z 1038.691,A -85,B 0,C 180,E1 -12068.187,E2 -12068.187} C_VEL
LIN {X 0,Y 382.952,Z 1031.313,A -85,B 0,C 180,E1 -12069.508,E2 -12069.508} C_VEL
LIN {X 0,Y 383.375,Z 1023.962,A -85,B 0,C 180,E1 -12070.564,E2 -12070.564} C_VEL
LIN {X 0,Y 383.836,Z 1016.148,A -85,B 0,C 180,E1 -12071.486,E2 -12071.486} C_VEL
LIN {X 0,Y 384.236,Z 1007.964,A -85,B 0,C 180,E1 -12072.277,E2 -12072.277} C_VEL
LIN {X 0,Y 384.639,Z 999.53,A -85,B 0,C 180,E1 -12072.935,E2 -12072.935} C_VEL
LIN {X 0,Y 385.029,Z 988.641,A -85,B 0,C 180,E1 -12073.593,E2 -12073.593} C_VEL
LIN {X 0,Y 385.37,Z 977.351,A -85,B 0,C 180,E1 -12074.051,E2 -12074.051} C_VEL
LIN {X 0,Y 385.855,Z 949.613,A -85,B 0,C 180,E1 -12074.707,E2 -12074.707} C_VEL
LIN {X 0,Y 386.317,Z 916.969,A -85,B 0,C 180,E1 -12075.453,E2 -12075.453} C_VEL
LIN {X 0,Y 383.302,Z 899.023,A -85,B 0,C 180,E1 -12075.999,E2 -12075.999} C_VEL
LIN {X 0,Y 383.554,Z 892.044,A -85,B 0,C 180,E1 -12078.15,E2 -12078.15} C_VEL
LIN {X 0,Y 383.115,Z 887.572,A -85,B 0,C 180,E1 -12079.63,E2 -12079.63} C_VEL
LIN {X 0,Y 383.005,Z 887.585,A -85,B 0,C 180,E1 -12083.81,E2 -12083.81} C_VEL
LIN {X 0,Y 382.966,Z 887.596,A -85,B 0,C 180,E1 -12087.31,E2 -12087.31} C_VEL
LIN {X 0,Y 382.98,Z 887.59,A -85,B 0,C 180,E1 -12090.92,E2 -12090.92} C_VEL
LIN {X 0,Y 383.014,Z 887.584,A -85,B 0,C 180,E1 -12094.669,E2 -12094.669} C_VEL
LIN {X 0,Y 382.993,Z 887.591,A -85,B 0,C 180,E1 -12097.902,E2 -12097.902} C_VEL
LIN {X 0,Y 382.962,Z 887.592,A -85,B 0,C 180,E1 -12101.351,E2 -12101.351} C_VEL
LIN {X 0,Y 382.99,Z 887.59,A -85,B 0,C 180,E1 -12104.303,E2 -12104.303} C_VEL
LIN {X 0,Y 382.984,Z 887.588,A -85,B 0,C 180,E1 -12107.237,E2 -12107.237} C_VEL
LIN {X 0,Y 382.986,Z 887.593,A -85,B 0,C 180,E1 -12110.42,E2 -12110.42} C_VEL
LIN {X 0,Y 383.018,Z 887.586,A -85,B 0,C 180,E1 -12114.044,E2 -12114.044} C_VEL
LIN {X 0,Y 382.986,Z 887.587,A -85,B 0,C 180,E1 -12117.58,E2 -12117.58} C_VEL
LIN {X 0,Y 382.976,Z 887.591,A -85,B 0,C 180,E1 -12120.299,E2 -12120.299} C_VEL
LIN {X 0,Y 383.006,Z 887.585,A -85,B 0,C 180,E1 -12124.046,E2 -12124.046} C_VEL
LIN {X 0,Y 382.988,Z 887.59,A -85,B 0,C 180,E1 -12127.334,E2 -12127.334} C_VEL
LIN {X 0,Y 383.023,Z 887.585,A -85,B 0,C 180,E1 -12130.714,E2 -12130.714} C_VEL
LIN {X 0,Y 383.074,Z 887.577,A -85,B 0,C 180,E1 -12134.027,E2 -12134.027} C_VEL
LIN {X 0,Y 383.137,Z 887.573,A -85,B 0,C 180,E1 -12137.284,E2 -12137.284} C_VEL
LIN {X 0,Y 383.139,Z 887.568,A -85,B 0,C 180,E1 -12140.498,E2 -12140.498} C_VEL
LIN {X 0,Y 383.237,Z 887.562,A -85,B 0,C 180,E1 -12143.683,E2 -12143.683} C_VEL
LIN {X 0,Y 383.368,Z 887.546,A -85,B 0,C 180,E1 -12147.899,E2 -12147.899} C_VEL
LIN {X 0,Y 383.264,Z 887.552,A -85,B 0,C 180,E1 -12151.051,E2 -12151.051} C_VEL
LIN {X 0,Y 383.367,Z 887.546,A -85,B 0,C 180,E1 -12152.101,E2 -12152.101} C_VEL
LIN {X 0,Y 383.238,Z 887.563,A -85,B 0,C 180,E1 -12156.317,E2 -12156.317} C_VEL
LIN {X 0,Y 383.139,Z 887.568,A -85,B 0,C 180,E1 -12159.503,E2 -12159.503} C_VEL
LIN {X 0,Y 383.134,Z 887.569,A -85,B 0,C 180,E1 -12163.538,E2 -12163.538} C_VEL
LIN {X 0,Y 383.058,Z 887.579,A -85,B 0,C 180,E1 -12167.434,E2 -12167.434} C_VEL
LIN {X 0,Y 383.019,Z 887.586,A -85,B 0,C 180,E1 -12170.641,E2 -12170.641} C_VEL
LIN {X 0,Y 383.008,Z 887.585,A -85,B 0,C 180,E1 -12173.809,E2 -12173.809} C_VEL
LIN {X 0,Y 382.979,Z 887.59,A -85,B 0,C 180,E1 -12174.721,E2 -12174.721} C_VEL
LIN {X 0,Y 382.327,Z 887.678,A -85,B 0,C 180,E1 -12175.599,E2 -12175.599} C_VEL
LIN {X 0,Y 379.465,Z 888.038,A -85,B 0,C 180,E1 -12177.025,E2 -12177.025} C_VEL
LIN {X 0,Y 377.034,Z 888.338,A -85,B 0,C 180,E1 -12178.178,E2 -12178.178} C_VEL
LIN {X 0,Y 375.994,Z 888.462,A -85,B 0,C 180,E1 -12179.071,E2 -12179.071} C_VEL
LIN {X 0,Y 375.912,Z 888.469,A -85,B 0,C 180,E1 -12179.373,E2 -12179.373} C_VEL
LIN {X 0,Y 375.951,Z 888.464,A -85,B 0,C 180,E1 -12182.829,E2 -12182.829} C_VEL
LIN {X 0,Y 375.952,Z 888.468,A -85,B 0,C 180,E1 -12185.416,E2 -12185.416} C_VEL
LIN {X 0,Y 375.937,Z 888.467,A -85,B 0,C 180,E1 -12188.262,E2 -12188.262} C_VEL
LIN {X 0,Y 375.917,Z 888.471,A -85,B 0,C 180,E1 -12191.597,E2 -12191.597} C_VEL
LIN {X 0,Y 375.923,Z 888.467,A -85,B 0,C 180,E1 -12194.73,E2 -12194.73} C_VEL
LIN {X 0,Y 375.911,Z 888.471,A -85,B 0,C 180,E1 -12197.696,E2 -12197.696} C_VEL
LIN {X 0,Y 375.936,Z 888.469,A -85,B 0,C 180,E1 -12200.533,E2 -12200.533} C_VEL
LIN {X 0,Y 375.961,Z 888.462,A -85,B 0,C 180,E1 -12203.497,E2 -12203.497} C_VEL
LIN {X 0,Y 375.961,Z 888.463,A -85,B 0,C 180,E1 -12205.888,E2 -12205.888} C_VEL
LIN {X 0,Y 375.963,Z 888.462,A -85,B 0,C 180,E1 -12209.687,E2 -12209.687} C_VEL
LIN {X 0,Y 375.919,Z 888.468,A -85,B 0,C 180,E1 -12212.134,E2 -12212.134} C_VEL
LIN {X 0,Y 375.937,Z 888.468,A -85,B 0,C 180,E1 -12214.533,E2 -12214.533} C_VEL
LIN {X 0,Y 375.971,Z 888.466,A -85,B 0,C 180,E1 -12216.886,E2 -12216.886} C_VEL
LIN {X 0,Y 375.967,Z 888.462,A -85,B 0,C 180,E1 -12220.337,E2 -12220.337} C_VEL
LIN {X 0,Y 375.972,Z 888.463,A -85,B 0,C 180,E1 -12223.716,E2 -12223.716} C_VEL
LIN {X 0,Y 376.102,Z 888.447,A -85,B 0,C 180,E1 -12227.041,E2 -12227.041} C_VEL
LIN {X 0,Y 376.108,Z 888.444,A -85,B 0,C 180,E1 -12230.318,E2 -12230.318} C_VEL
LIN {X 0,Y 376.195,Z 888.438,A -85,B 0,C 180,E1 -12233.564,E2 -12233.564} C_VEL
LIN {X 0,Y 376.329,Z 888.422,A -85,B 0,C 180,E1 -12237.859,E2 -12237.859} C_VEL
LIN {X 0,Y 376.233,Z 888.428,A -85,B 0,C 180,E1 -12241.07,E2 -12241.07} C_VEL
LIN {X 0,Y 376.329,Z 888.423,A -85,B 0,C 180,E1 -12242.14,E2 -12242.14} C_VEL
LIN {X 0,Y 376.195,Z 888.439,A -85,B 0,C 180,E1 -12246.435,E2 -12246.435} C_VEL
LIN {X 0,Y 376.107,Z 888.444,A -85,B 0,C 180,E1 -12249.681,E2 -12249.681} C_VEL
LIN {X 0,Y 376.093,Z 888.446,A -85,B 0,C 180,E1 -12253.658,E2 -12253.658} C_VEL
LIN {X 0,Y 376.008,Z 888.456,A -85,B 0,C 180,E1 -12257.588,E2 -12257.588} C_VEL
LIN {X 0,Y 375.98,Z 888.465,A -85,B 0,C 180,E1 -12260.832,E2 -12260.832} C_VEL
LIN {X 0,Y 375.932,Z 888.466,A -85,B 0,C 180,E1 -12264.285,E2 -12264.285} C_VEL
LIN {X 0,Y 375.91,Z 888.47,A -85,B 0,C 180,E1 -12266.66,E2 -12266.66} C_VEL
LIN {X 0,Y 375.912,Z 888.472,A -85,B 0,C 180,E1 -12269.084,E2 -12269.084} C_VEL
LIN {X 0,Y 375.953,Z 888.469,A -85,B 0,C 180,E1 -12271.562,E2 -12271.562} C_VEL
LIN {X 0,Y 375.948,Z 888.469,A -85,B 0,C 180,E1 -12275.416,E2 -12275.416} C_VEL
LIN {X 0,Y 375.933,Z 888.467,A -85,B 0,C 180,E1 -12278.262,E2 -12278.262} C_VEL
LIN {X 0,Y 375.912,Z 888.472,A -85,B 0,C 180,E1 -12281.596,E2 -12281.596} C_VEL
LIN {X 0,Y 375.919,Z 888.468,A -85,B 0,C 180,E1 -12284.73,E2 -12284.73} C_VEL
LIN {X 0,Y 375.906,Z 888.471,A -85,B 0,C 180,E1 -12287.696,E2 -12287.696} C_VEL
LIN {X 0,Y 375.931,Z 888.47,A -85,B 0,C 180,E1 -12290.533,E2 -12290.533} C_VEL
LIN {X 0,Y 375.957,Z 888.463,A -85,B 0,C 180,E1 -12293.497,E2 -12293.497} C_VEL
LIN {X 0,Y 375.957,Z 888.464,A -85,B 0,C 180,E1 -12295.888,E2 -12295.888} C_VEL
LIN {X 0,Y 375.958,Z 888.462,A -85,B 0,C 180,E1 -12299.686,E2 -12299.686} C_VEL
LIN {X 0,Y 376.012,Z 888.632,A -85,B 0,C 180,E1 -12303.475,E2 -12303.475} C_VEL
LIN {X 0,Y 378.033,Z 899.537,A -85,B 0,C 180,E1 -12306.44,E2 -12306.44} C_VEL
LIN {X 0,Y 378.029,Z 904.007,A -85,B 0,C 180,E1 -12307.597,E2 -12307.597} C_VEL
LIN {X 0,Y 376.952,Z 918.444,A -85,B 0,C 180,E1 -12311.239,E2 -12311.239} C_VEL
LIN {X 0,Y 376.275,Z 928.608,A -85,B 0,C 180,E1 -12313.778,E2 -12313.778} C_VEL
LIN {X 0,Y 379.208,Z 955.341,A -85,B 0,C 180,E1 -12314.521,E2 -12314.521} C_VEL
LIN {X 0,Y 378.39,Z 1006.927,A -85,B 0,C 180,E1 -12315.753,E2 -12315.753} C_VEL
LIN {X 0,Y 377.838,Z 1018.593,A -85,B 0,C 180,E1 -12316.212,E2 -12316.212} C_VEL
LIN {X 0,Y 377.486,Z 1028.711,A -85,B 0,C 180,E1 -12316.816,E2 -12316.816} C_VEL
LIN {X 0,Y 377.031,Z 1037.38,A -85,B 0,C 180,E1 -12317.485,E2 -12317.485} C_VEL
LIN {X 0,Y 376.526,Z 1045.73,A -85,B 0,C 180,E1 -12318.288,E2 -12318.288} C_VEL
LIN {X 0,Y 376.07,Z 1053.687,A -85,B 0,C 180,E1 -12319.229,E2 -12319.229} C_VEL
LIN {X 0,Y 375.577,Z 1061.144,A -85,B 0,C 180,E1 -12320.304,E2 -12320.304} C_VEL
LIN {X 0,Y 375.152,Z 1068.7,A -85,B 0,C 180,E1 -12321.652,E2 -12321.652} C_VEL
LIN {X 0,Y 374.947,Z 1074.578,A -85,B 0,C 180,E1 -12323.002,E2 -12323.002} C_VEL
LIN {X 0,Y 374.679,Z 1078.559,A -85,B 0,C 180,E1 -12324.128,E2 -12324.128} C_VEL
LIN {X 0,Y 374.682,Z 1081.543,A -85,B 0,C 180,E1 -12325.158,E2 -12325.158} C_VEL
LIN {X 0,Y 374.519,Z 1084.927,A -85,B 0,C 180,E1 -12326.773,E2 -12326.773} C_VEL
LIN {X 0,Y 374.549,Z 1086.53,A -85,B 0,C 180,E1 -12327.849,E2 -12327.849} C_VEL
LIN {X 0,Y 374.604,Z 1087.513,A -85,B 0,C 180,E1 -12328.925,E2 -12328.925} C_VEL
LIN {X 0,Y 374.586,Z 1087.904,A -85,B 0,C 180,E1 -12330,E2 -12330} C_VEL
LIN {X 0,Y 374.582,Z 1087.781,A -85,B 0,C 180,E1 -12331.075,E2 -12331.075} C_VEL
LIN {X 0,Y 374.512,Z 1087.142,A -85,B 0,C 180,E1 -12332.151,E2 -12332.151} C_VEL
LIN {X 0,Y 374.51,Z 1085.981,A -85,B 0,C 180,E1 -12333.227,E2 -12333.227} C_VEL
LIN {X 0,Y 374.657,Z 1083.066,A -85,B 0,C 180,E1 -12334.842,E2 -12334.842} C_VEL
LIN {X 0,Y 374.764,Z 1079.233,A -85,B 0,C 180,E1 -12336.326,E2 -12336.326} C_VEL
LIN {X 0,Y 375.01,Z 1075.165,A -85,B 0,C 180,E1 -12337.538,E2 -12337.538} C_VEL
LIN {X 0,Y 375.376,Z 1069.505,A -85,B 0,C 180,E1 -12338.885,E2 -12338.885} C_VEL
LIN {X 0,Y 375.938,Z 1062.461,A -85,B 0,C 180,E1 -12340.23,E2 -12340.23} C_VEL
LIN {X 0,Y 376.696,Z 1053.409,A -85,B 0,C 180,E1 -12341.57,E2 -12341.57} C_VEL
LIN {X 0,Y 377.281,Z 1045.557,A -85,B 0,C 180,E1 -12342.506,E2 -12342.506} C_VEL
LIN {X 0,Y 377.854,Z 1037.439,A -85,B 0,C 180,E1 -12343.307,E2 -12343.307} C_VEL
LIN {X 0,Y 378.395,Z 1029.153,A -85,B 0,C 180,E1 -12343.972,E2 -12343.972} C_VEL
LIN {X 0,Y 379.046,Z 1019.717,A -85,B 0,C 180,E1 -12344.564,E2 -12344.564} C_VEL
LIN {X 0,Y 379.764,Z 1007.067,A -85,B 0,C 180,E1 -12345.124,E2 -12345.124} C_VEL
LIN {X 0,Y 380.631,Z 971.652,A -85,B 0,C 180,E1 -12346.043,E2 -12346.043} C_VEL
LIN {X 0,Y 380.962,Z 953.735,A -85,B 0,C 180,E1 -12346.512,E2 -12346.512} C_VEL
LIN {X 0,Y 379.34,Z 939.281,A -85,B 0,C 180,E1 -12347.028,E2 -12347.028} C_VEL
LIN {X 0,Y 376.925,Z 926.264,A -85,B 0,C 180,E1 -12347.592,E2 -12347.592} C_VEL
LIN {X 0,Y 378.376,Z 911.171,A -85,B 0,C 180,E1 -12351.61,E2 -12351.61} C_VEL
LIN {X 0,Y 378.967,Z 904.428,A -85,B 0,C 180,E1 -12353.498,E2 -12353.498} C_VEL
LIN {X 0,Y 378.162,Z 898.623,A -85,B 0,C 180,E1 -12355.305,E2 -12355.305} C_VEL
LIN {X 0,Y 376.347,Z 890.234,A -85,B 0,C 180,E1 -12358.184,E2 -12358.184} C_VEL
LIN {X 0,Y 375.927,Z 888.473,A -85,B 0,C 180,E1 -12358.916,E2 -12358.916} C_VEL
LIN {X 0,Y 375.952,Z 888.471,A -85,B 0,C 180,E1 -12361.562,E2 -12361.562} C_VEL
LIN {X 0,Y 375.946,Z 888.47,A -85,B 0,C 180,E1 -12365.417,E2 -12365.417} C_VEL
LIN {X 0,Y 375.929,Z 888.471,A -85,B 0,C 180,E1 -12368.262,E2 -12368.262} C_VEL
LIN {X 0,Y 375.91,Z 888.475,A -85,B 0,C 180,E1 -12371.597,E2 -12371.597} C_VEL
LIN {X 0,Y 375.917,Z 888.471,A -85,B 0,C 180,E1 -12374.73,E2 -12374.73} C_VEL
LIN {X 0,Y 375.904,Z 888.473,A -85,B 0,C 180,E1 -12377.696,E2 -12377.696} C_VEL
LIN {X 0,Y 375.93,Z 888.47,A -85,B 0,C 180,E1 -12380.534,E2 -12380.534} C_VEL
LIN {X 0,Y 375.954,Z 888.466,A -85,B 0,C 180,E1 -12383.498,E2 -12383.498} C_VEL
LIN {X 0,Y 375.955,Z 888.467,A -85,B 0,C 180,E1 -12385.889,E2 -12385.889} C_VEL
LIN {X 0,Y 375.958,Z 888.466,A -85,B 0,C 180,E1 -12389.687,E2 -12389.687} C_VEL
LIN {X 0,Y 375.914,Z 888.473,A -85,B 0,C 180,E1 -12392.135,E2 -12392.135} C_VEL
LIN {X 0,Y 375.932,Z 888.474,A -85,B 0,C 180,E1 -12394.534,E2 -12394.534} C_VEL
LIN {X 0,Y 375.984,Z 888.665,A -85,B 0,C 180,E1 -12397.179,E2 -12397.179} C_VEL
LIN {X 0,Y 377.267,Z 894.966,A -85,B 0,C 180,E1 -12399.841,E2 -12399.841} C_VEL
LIN {X 0,Y 377.725,Z 899.534,A -85,B 0,C 180,E1 -12401.607,E2 -12401.607} C_VEL
LIN {X 0,Y 377.591,Z 902.215,A -85,B 0,C 180,E1 -12402.553,E2 -12402.553} C_VEL
LIN {X 0,Y 381.257,Z 916.825,A -85,B 0,C 180,E1 -12403.242,E2 -12403.242} C_VEL
LIN {X 0,Y 381.659,Z 920.849,A -85,B 0,C 180,E1 -12403.385,E2 -12403.385} C_VEL
LIN {X 0,Y 380.012,Z 979.089,A -85,B 0,C 180,E1 -12404.908,E2 -12404.908} C_VEL
LIN {X 0,Y 379.559,Z 991.463,A -85,B 0,C 180,E1 -12405.456,E2 -12405.456} C_VEL
LIN {X 0,Y 378.97,Z 1000.899,A -85,B 0,C 180,E1 -12406.05,E2 -12406.05} C_VEL
LIN {X 0,Y 378.504,Z 1009.133,A -85,B 0,C 180,E1 -12406.717,E2 -12406.717} C_VEL
LIN {X 0,Y 377.996,Z 1017.151,A -85,B 0,C 180,E1 -12407.518,E2 -12407.518} C_VEL
LIN {X 0,Y 377.399,Z 1024.838,A -85,B 0,C 180,E1 -12408.452,E2 -12408.452} C_VEL
LIN {X 0,Y 376.662,Z 1033.731,A -85,B 0,C 180,E1 -12409.79,E2 -12409.79} C_VEL
LIN {X 0,Y 376.032,Z 1040.613,A -85,B 0,C 180,E1 -12411.131,E2 -12411.131} C_VEL
LIN {X 0,Y 375.759,Z 1044.144,A -85,B 0,C 180,E1 -12411.937,E2 -12411.937} C_VEL
LIN {X 0,Y 375.36,Z 1049.65,A -85,B 0,C 180,E1 -12413.55,E2 -12413.55} C_VEL
LIN {X 0,Y 374.926,Z 1053.709,A -85,B 0,C 180,E1 -12415.162,E2 -12415.162} C_VEL
LIN {X 0,Y 374.835,Z 1056.448,A -85,B 0,C 180,E1 -12416.776,E2 -12416.776} C_VEL
LIN {X 0,Y 374.722,Z 1057.503,A -85,B 0,C 180,E1 -12417.851,E2 -12417.851} C_VEL
LIN {X 0,Y 374.614,Z 1058.051,A -85,B 0,C 180,E1 -12418.926,E2 -12418.926} C_VEL
LIN {X 0,Y 374.588,Z 1058.094,A -85,B 0,C 180,E1 -12420,E2 -12420} C_VEL
LIN {X 0,Y 374.593,Z 1057.627,A -85,B 0,C 180,E1 -12421.076,E2 -12421.076} C_VEL
LIN {X 0,Y 374.614,Z 1056.566,A -85,B 0,C 180,E1 -12422.151,E2 -12422.151} C_VEL
LIN {X 0,Y 374.666,Z 1053.934,A -85,B 0,C 180,E1 -12423.765,E2 -12423.765} C_VEL
LIN {X 0,Y 374.804,Z 1051.462,A -85,B 0,C 180,E1 -12424.841,E2 -12424.841} C_VEL
LIN {X 0,Y 375.045,Z 1046.435,A -85,B 0,C 180,E1 -12426.456,E2 -12426.456} C_VEL
LIN {X 0,Y 375.319,Z 1040.992,A -85,B 0,C 180,E1 -12427.803,E2 -12427.803} C_VEL
LIN {X 0,Y 375.606,Z 1035.647,A -85,B 0,C 180,E1 -12428.881,E2 -12428.881} C_VEL
LIN {X 0,Y 376.045,Z 1029.206,A -85,B 0,C 180,E1 -12429.956,E2 -12429.956} C_VEL
LIN {X 0,Y 376.519,Z 1021.386,A -85,B 0,C 180,E1 -12431.031,E2 -12431.031} C_VEL
LIN {X 0,Y 377.065,Z 1011.643,A -85,B 0,C 180,E1 -12432.104,E2 -12432.104} C_VEL
LIN {X 0,Y 377.534,Z 1002.145,A -85,B 0,C 180,E1 -12432.909,E2 -12432.909} C_VEL
LIN {X 0,Y 377.903,Z 993.067,A -85,B 0,C 180,E1 -12433.511,E2 -12433.511} C_VEL
LIN {X 0,Y 378.098,Z 983.721,A -85,B 0,C 180,E1 -12433.984,E2 -12433.984} C_VEL
LIN {X 0,Y 378.463,Z 973.141,A -85,B 0,C 180,E1 -12434.347,E2 -12434.347} C_VEL
LIN {X 0,Y 379.363,Z 917.864,A -85,B 0,C 180,E1 -12435.641,E2 -12435.641} C_VEL
LIN {X 0,Y 376.308,Z 899.307,A -85,B 0,C 180,E1 -12436.211,E2 -12436.211} C_VEL
LIN {X 0,Y 376.541,Z 893.425,A -85,B 0,C 180,E1 -12438.052,E2 -12438.052} C_VEL
LIN {X 0,Y 376.075,Z 888.449,A -85,B 0,C 180,E1 -12439.728,E2 -12439.728} C_VEL
LIN {X 0,Y 375.968,Z 888.463,A -85,B 0,C 180,E1 -12443.658,E2 -12443.658} C_VEL
LIN {X 0,Y 375.91,Z 888.47,A -85,B 0,C 180,E1 -12446.661,E2 -12446.661} C_VEL
LIN {X 0,Y 375.913,Z 888.472,A -85,B 0,C 180,E1 -12449.085,E2 -12449.085} C_VEL
LIN {X 0,Y 375.956,Z 888.468,A -85,B 0,C 180,E1 -12451.563,E2 -12451.563} C_VEL
LIN {X 0,Y 375.952,Z 888.468,A -85,B 0,C 180,E1 -12455.417,E2 -12455.417} C_VEL
LIN {X 0,Y 375.935,Z 888.467,A -85,B 0,C 180,E1 -12458.263,E2 -12458.263} C_VEL
LIN {X 0,Y 375.915,Z 888.472,A -85,B 0,C 180,E1 -12461.597,E2 -12461.597} C_VEL
LIN {X 0,Y 375.922,Z 888.468,A -85,B 0,C 180,E1 -12464.731,E2 -12464.731} C_VEL
LIN {X 0,Y 375.909,Z 888.471,A -85,B 0,C 180,E1 -12467.697,E2 -12467.697} C_VEL
LIN {X 0,Y 375.934,Z 888.469,A -85,B 0,C 180,E1 -12470.534,E2 -12470.534} C_VEL
LIN {X 0,Y 375.96,Z 888.462,A -85,B 0,C 180,E1 -12473.497,E2 -12473.497} C_VEL
LIN {X 0,Y 375.961,Z 888.464,A -85,B 0,C 180,E1 -12475.889,E2 -12475.889} C_VEL
LIN {X 0,Y 375.963,Z 888.462,A -85,B 0,C 180,E1 -12479.687,E2 -12479.687} C_VEL
LIN {X 0,Y 375.919,Z 888.469,A -85,B 0,C 180,E1 -12482.135,E2 -12482.135} C_VEL
LIN {X 0,Y 375.97,Z 888.461,A -85,B 0,C 180,E1 -12485.717,E2 -12485.717} C_VEL
LIN {X 0,Y 375.961,Z 888.468,A -85,B 0,C 180,E1 -12489.196,E2 -12489.196} C_VEL
LIN {X 0,Y 376.017,Z 888.456,A -85,B 0,C 180,E1 -12492.6,E2 -12492.6} C_VEL
LIN {X 0,Y 376.094,Z 888.446,A -85,B 0,C 180,E1 -12496.343,E2 -12496.343} C_VEL
LIN {X 0,Y 376.11,Z 888.444,A -85,B 0,C 180,E1 -12500.318,E2 -12500.318} C_VEL
LIN {X 0,Y 376.197,Z 888.437,A -85,B 0,C 180,E1 -12503.564,E2 -12503.564} C_VEL
LIN {X 0,Y 376.332,Z 888.422,A -85,B 0,C 180,E1 -12507.86,E2 -12507.86} C_VEL
LIN {X 0,Y 376.235,Z 888.428,A -85,B 0,C 180,E1 -12511.071,E2 -12511.071} C_VEL
LIN {X 0,Y 376.331,Z 888.423,A -85,B 0,C 180,E1 -12512.141,E2 -12512.141} C_VEL
LIN {X 0,Y 376.197,Z 888.438,A -85,B 0,C 180,E1 -12516.436,E2 -12516.436} C_VEL
LIN {X 0,Y 376.11,Z 888.444,A -85,B 0,C 180,E1 -12519.682,E2 -12519.682} C_VEL
LIN {X 0,Y 376.096,Z 888.445,A -85,B 0,C 180,E1 -12523.658,E2 -12523.658} C_VEL
LIN {X 0,Y 376.011,Z 888.456,A -85,B 0,C 180,E1 -12527.589,E2 -12527.589} C_VEL
LIN {X 0,Y 375.984,Z 888.465,A -85,B 0,C 180,E1 -12530.832,E2 -12530.832} C_VEL
LIN {X 0,Y 375.936,Z 888.466,A -85,B 0,C 180,E1 -12534.286,E2 -12534.286} C_VEL
LIN {X 0,Y 375.913,Z 888.47,A -85,B 0,C 180,E1 -12536.661,E2 -12536.661} C_VEL
LIN {X 0,Y 375.912,Z 888.469,A -85,B 0,C 180,E1 -12539.373,E2 -12539.373} C_VEL
LIN {X 0,Y 375.251,Z 888.551,A -85,B 0,C 180,E1 -12540.268,E2 -12540.268} C_VEL
LIN {X 0,Y 372.399,Z 888.909,A -85,B 0,C 180,E1 -12541.722,E2 -12541.722} C_VEL
LIN {X 0,Y 369.989,Z 889.211,A -85,B 0,C 180,E1 -12542.899,E2 -12542.899} C_VEL
LIN {X 0,Y 368.967,Z 889.338,A -85,B 0,C 180,E1 -12543.809,E2 -12543.809} C_VEL
LIN {X 0,Y 368.89,Z 889.344,A -85,B 0,C 180,E1 -12544.117,E2 -12544.117} C_VEL
LIN {X 0,Y 368.898,Z 889.347,A -85,B 0,C 180,E1 -12547.564,E2 -12547.564} C_VEL
LIN {X 0,Y 368.887,Z 889.345,A -85,B 0,C 180,E1 -12550.374,E2 -12550.374} C_VEL
LIN {X 0,Y 368.882,Z 889.347,A -85,B 0,C 180,E1 -12553.615,E2 -12553.615} C_VEL
LIN {X 0,Y 368.887,Z 889.344,A -85,B 0,C 180,E1 -12556.695,E2 -12556.695} C_VEL
LIN {X 0,Y 368.888,Z 889.345,A -85,B 0,C 180,E1 -12559.648,E2 -12559.648} C_VEL
LIN {X 0,Y 368.899,Z 889.342,A -85,B 0,C 180,E1 -12563.145,E2 -12563.145} C_VEL
